KUKA KRL program: MyProgram_099().src

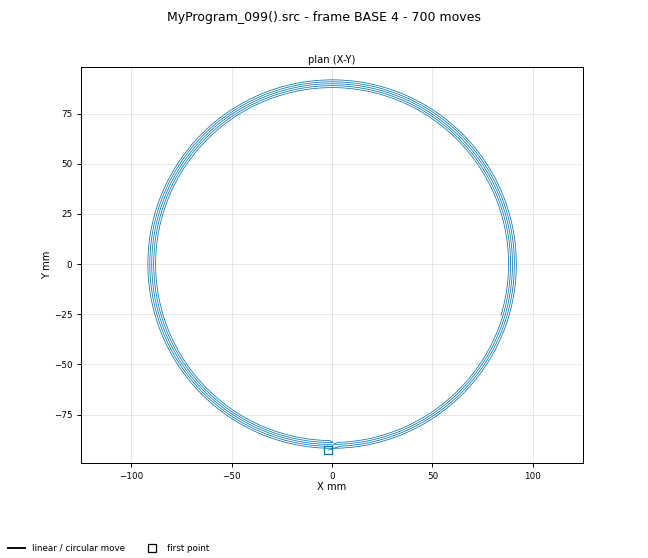
[picture p0: tool path of MyProgram_099().src in frame BASE 4, 700 of 700 moves have a stored position in this frame; points joined in program order, loops and branches not executed]
&ACCESS RVP
&REL 1
&PARAM TEMPLATE = C:\KRC\Roboter\Template\vorgabe
&PARAM EDITMASK = *
DEF MyProgram_099()
; ---- Setting reference (Base) ----
$BASE = BASE_DATA[4]

; --------------------------
; ---- Setting tool (TCP) ----
$TOOL = TOOL_DATA[3]
; --------------------------

$VEL.CP = VEL_APROX_PRINT
Startdeposition()
$VEL.CP = VEL_PRINT
LIN {X -1.871,Y -92.7683,Z 91,A -94.8232,B 24.9323,C -1.9,E1 24.9994,E2 179.961} C_DIS
Enddeposition()
LIN {X 0.618,Y -91.7983,Z 91,A -93.6423,B 24.932,C -1.905,E1 25.0028,E2 178.7684} C_DIS
Startdeposition()
$VEL.CP = VEL_PRINT
LIN {X -1.6204,Y -91.8049,Z 91,A -96.9281,B 24.9365,C -1.8408,E1 24.9932,E2 182.2064} C_DIS
LIN {X -6.6476,Y -91.5793,Z 91,A -99.0466,B 24.9341,C -1.8746,E1 24.9875,E2 184.2456} C_DIS
LIN {X -12.2271,Y -91.0017,Z 91,A -103.2009,B 24.9356,C -1.8535,E1 24.9758,E2 188.4527} C_DIS
LIN {X -15.9011,Y -90.4321,Z 91,A -104.6147,B 24.9335,C -1.8841,E1 24.9721,E2 189.7952} C_DIS
LIN {X -18.2695,Y -89.9835,Z 91,A -106.7072,B 24.9348,C -1.8652,E1 24.9662,E2 191.9348} C_DIS
LIN {X -22.9812,Y -88.8968,Z 91,A -109.6487,B 24.9345,C -1.8693,E1 24.9583,E2 194.8706} C_DIS
LIN {X -27.0599,Y -87.7413,Z 91,A -111.9748,B 24.9336,C -1.8816,E1 24.9521,E2 197.1715} C_DIS
LIN {X -31.2211,Y -86.3485,Z 91,A -114.7916,B 24.9336,C -1.8813,E1 24.9447,E2 199.9944} C_DIS
LIN {X -34.2722,Y -85.1832,Z 91,A -116.9435,B 24.9338,C -1.8795,E1 24.939,E2 202.1551} C_DIS
LIN {X -37.6537,Y -83.7434,Z 91,A -119.5434,B 24.9343,C -1.8722,E1 24.9323,E2 204.7786} C_DIS
LIN {X -42.2252,Y -81.5349,Z 91,A -122.8582,B 24.9343,C -1.8714,E1 24.9241,E2 208.1042} C_DIS
LIN {X -45.2073,Y -79.9207,Z 91,A -124.3084,B 24.9326,C -1.8955,E1 24.9206,E2 209.5014} C_DIS
LIN {X -48.7304,Y -77.8211,Z 91,A -127.0637,B 24.9328,C -1.893,E1 24.914,E2 212.271} C_DIS
LIN {X -51.619,Y -75.9359,Z 91,A -129.5861,B 24.9334,C -1.8847,E1 24.9081,E2 214.8214} C_DIS
LIN {X -54.5175,Y -73.8832,Z 91,A -131.4951,B 24.9325,C -1.8981,E1 24.9039,E2 216.7051} C_DIS
LIN {X -58.7556,Y -70.5588,Z 91,A -134.6797,B 24.9316,C -1.9098,E1 24.8969,E2 219.8739} C_DIS
LIN {X -60.9727,Y -68.6527,Z 91,A -136.6778,B 24.9318,C -1.9079,E1 24.8927,E2 221.8844} C_DIS
LIN {X -64.9121,Y -64.9421,Z 91,A -140.0394,B 24.9312,C -1.9153,E1 24.8859,E2 225.2422} C_DIS
LIN {X -67.1815,Y -62.5906,Z 91,A -142.1304,B 24.931,C -1.9181,E1 24.8819,E2 227.3356} C_DIS
LIN {X -70.739,Y -58.5387,Z 91,A -145.139,B 24.9297,C -1.9368,E1 24.8765,E2 230.3132} C_DIS
LIN {X -72.1644,Y -56.7724,Z 91,A -146.9681,B 24.9304,C -1.9274,E1 24.8732,E2 232.1734} C_DIS
LIN {X -75.8177,Y -51.7933,Z 91,A -150.4821,B 24.9289,C -1.9474,E1 24.8675,E2 235.657} C_DIS
LIN {X -77.8299,Y -48.7162,Z 91,A -153.8723,B 24.9309,C -1.92,E1 24.8623,E2 239.1296} C_DIS
LIN {X -80.0718,Y -44.9366,Z 91,A -155.5096,B 24.9279,C -1.9607,E1 24.8602,E2 240.6782} C_DIS
LIN {X -82.9877,Y -39.291,Z 91,A -159.9053,B 24.9281,C -1.9585,E1 24.8546,E2 245.1028} C_DIS
LIN {X -84.5445,Y -35.8192,Z 91,A -162.2753,B 24.9276,C -1.9654,E1 24.8519,E2 247.4694} C_DIS
LIN {X -86.3463,Y -31.2273,Z 91,A -165.1608,B 24.9265,C -1.9802,E1 24.8491,E2 250.3359} C_DIS
LIN {X -87.3543,Y -28.2838,Z 91,A -167.9303,B 24.9279,C -1.9612,E1 24.8466,E2 253.1666} C_DIS
LIN {X -88.49,Y -24.5019,Z 91,A -169.5246,B 24.9254,C -1.9946,E1 24.8454,E2 254.6904} C_DIS
LIN {X -89.3909,Y -20.979,Z 91,A -172.0935,B 24.9256,C -1.9925,E1 24.8437,E2 257.2792} C_DIS
LIN {X -90.1571,Y -17.3912,Z 91,A -174.3422,B 24.9249,C -2.0008,E1 24.8424,E2 259.5214} C_DIS
LIN {X -90.8192,Y -13.5236,Z 91,A -176.8189,B 24.9244,C -2.0076,E1 24.8413,E2 261.9966} C_DIS
LIN {X -91.1749,Y -10.8598,Z 91,A -178.5376,B 24.9241,C -2.0117,E1 24.8407,E2 263.716} C_DIS
LIN {X -91.5267,Y -7.3223,Z 91,A 179.3238,B 24.9234,C -2.0211,E1 24.8402,E2 265.8449} C_DIS
LIN {X -91.7396,Y -3.824,Z 91,A 177.0719,B 24.923,C -2.0261,E1 24.8399,E2 268.0983} C_DIS
LIN {X -91.8155,Y -0.8782,Z 91,A 175.1478,B 24.9228,C -2.0294,E1 24.8398,E2 270.0261} C_DIS
LIN {X -91.7727,Y 2.9233,Z 91,A 172.771,B 24.9222,C -2.0369,E1 24.8399,E2 272.3994} C_DIS
LIN {X -91.5374,Y 7.1893,Z 91,A 169.952,B 24.9219,C -2.0409,E1 24.8404,E2 275.2257} C_DIS
LIN {X -91.1985,Y 10.6584,Z 91,A 167.9398,B 24.921,C -2.0527,E1 24.841,E2 277.2218} C_DIS
LIN {X -90.6942,Y 14.3323,Z 91,A 165.6777,B 24.9203,C -2.0617,E1 24.842,E2 279.4761} C_DIS
LIN {X -90.1147,Y 17.6113,Z 91,A 163.4344,B 24.9202,C -2.0634,E1 24.8431,E2 281.7286} C_DIS
LIN {X -88.9887,Y 22.6236,Z 91,A 160.5247,B 24.9187,C -2.0823,E1 24.8449,E2 284.6101} C_DIS
LIN {X -88.2612,Y 25.3131,Z 91,A 158.5023,B 24.9189,C -2.0793,E1 24.8465,E2 286.6515} C_DIS
LIN {X -86.9975,Y 29.3631,Z 91,A 155.3931,B 24.9193,C -2.0739,E1 24.8492,E2 289.7914} C_DIS
LIN {X -85.8688,Y 32.5163,Z 91,A 154.1404,B 24.9169,C -2.1052,E1 24.8503,E2 290.9765} C_DIS
LIN {X -85.0065,Y 34.7084,Z 91,A 151.2137,B 24.9199,C -2.0665,E1 24.8536,E2 294.0118} C_DIS
LIN {X -82.8239,Y 39.6354,Z 91,A 149.1226,B 24.9162,C -2.1142,E1 24.8559,E2 296.0005} C_DIS
LIN {X -81.6777,Y 41.947,Z 91,A 147.2257,B 24.9165,C -2.1103,E1 24.8583,E2 297.9169} C_DIS
LIN {X -79.0825,Y 46.6554,Z 91,A 143.9691,B 24.9155,C -2.123,E1 24.8627,E2 301.1604} C_DIS
LIN {X -76.1928,Y 51.2397,Z 91,A 140.5759,B 24.9147,C -2.1321,E1 24.8679,E2 304.549} C_DIS
LIN {X -73.3066,Y 55.2895,Z 91,A 137.3458,B 24.9144,C -2.1366,E1 24.8732,E2 307.7838} C_DIS
LIN {X -69.6332,Y 59.851,Z 91,A 134.0172,B 24.9128,C -2.156,E1 24.879,E2 311.0817} C_DIS
LIN {X -67.3029,Y 62.4597,Z 91,A 131.7335,B 24.9126,C -2.1584,E1 24.8833,E2 313.3699} C_DIS
LIN {X -65.444,Y 64.404,Z 91,A 129.8568,B 24.9128,C -2.1565,E1 24.8869,E2 315.2593} C_DIS
LIN {X -62.1113,Y 67.6236,Z 91,A 127.3843,B 24.9112,C -2.1761,E1 24.8918,E2 317.6952} C_DIS
LIN {X -59.1378,Y 70.2397,Z 91,A 124.4002,B 24.912,C -2.1659,E1 24.8982,E2 320.7153} C_DIS
LIN {X -56.3727,Y 72.4779,Z 91,A 121.6226,B 24.913,C -2.1536,E1 24.9044,E2 323.5324} C_DIS
LIN {X -53.4479,Y 74.6599,Z 91,A 119.949,B 24.9111,C -2.1767,E1 24.9081,E2 325.1569} C_DIS
LIN {X -49.435,Y 77.3756,Z 91,A 116.84,B 24.9109,C -2.1799,E1 24.9153,E2 328.2685} C_DIS
LIN {X -44.1429,Y 80.513,Z 91,A 113.2762,B 24.9096,C -2.1953,E1 24.9238,E2 331.8064} C_DIS
LIN {X -41.9976,Y 81.6518,Z 91,A 111.4688,B 24.9101,C -2.1887,E1 24.9283,E2 333.6345} C_DIS
LIN {X -38.7679,Y 83.2334,Z 91,A 108.7733,B 24.911,C -2.1781,E1 24.9352,E2 336.362} C_DIS
LIN {X -35.7147,Y 84.5885,Z 91,A 107.4169,B 24.9089,C -2.2039,E1 24.9386,E2 337.6602} C_DIS
LIN {X -31.6123,Y 86.2055,Z 91,A 104.5487,B 24.9089,C -2.2039,E1 24.9461,E2 340.5344} C_DIS
LIN {X -29.457,Y 86.9656,Z 91,A 102.41,B 24.9106,C -2.1832,E1 24.9518,E2 342.7265} C_DIS
LIN {X -25.9931,Y 88.0632,Z 91,A 100.6921,B 24.909,C -2.203,E1 24.9563,E2 344.4001} C_DIS
LIN {X -22.5168,Y 89.0161,Z 91,A 98.4003,B 24.9089,C -2.2039,E1 24.9625,E2 346.6932} C_DIS
LIN {X -17.696,Y 90.0984,Z 91,A 95.646,B 24.9078,C -2.2172,E1 24.9699,E2 349.4195} C_DIS
LIN {X -13.9628,Y 90.7513,Z 91,A 92.1983,B 24.9105,C -2.1842,E1 24.9797,E2 352.9488} C_DIS
LIN {X -9.5944,Y 91.3165,Z 91,A 90.3815,B 24.9079,C -2.2156,E1 24.9845,E2 354.692} C_DIS
LIN {X -7.0102,Y 91.5516,Z 91,A 87.5465,B 24.9111,C -2.1772,E1 24.9927,E2 357.6194} C_DIS
LIN {X -1.6648,Y 91.8041,Z 91,A 84.4297,B 24.9104,C -2.1852,E1 25.0013,E2 360.7175} C_DIS
LIN {X 2.9296,Y 91.7725,Z 91,A 82.8065,B 24.907,C -2.2261,E1 25.0056,E2 362.2432} C_DIS
LIN {X 5.2509,Y 91.6691,Z 91,A 80.5872,B 24.9091,C -2.2008,E1 25.0119,E2 364.5218} C_DIS
LIN {X 10.4898,Y 91.2182,Z 91,A 77.508,B 24.9086,C -2.2071,E1 25.0204,E2 367.5842} C_DIS
LIN {X 14.3424,Y 90.6926,Z 91,A 75.2122,B 24.9083,C -2.2107,E1 25.0267,E2 369.8692} C_DIS
LIN {X 17.7373,Y 90.0905,Z 91,A 73.0288,B 24.9085,C -2.2088,E1 25.0327,E2 372.0547} C_DIS
LIN {X 20.9469,Y 89.3984,Z 91,A 71.1006,B 24.9082,C -2.2118,E1 25.038,E2 373.9732} C_DIS
LIN {X 24.2742,Y 88.5526,Z 91,A 69.1138,B 24.9079,C -2.2157,E1 25.0433,E2 375.9477} C_DIS
LIN {X 28.1738,Y 87.39,Z 91,A 66.5053,B 24.9083,C -2.2115,E1 25.0503,E2 378.5616} C_DIS
LIN {X 31.0195,Y 86.4215,Z 91,A 64.3973,B 24.9091,C -2.202,E1 25.0559,E2 380.6879} C_DIS
LIN {X 34.6134,Y 85.0451,Z 91,A 61.6457,B 24.9102,C -2.1877,E1 25.0631,E2 383.4671} C_DIS
LIN {X 37.6375,Y 83.7507,Z 91,A 60.1052,B 24.909,C -2.2028,E1 25.0669,E2 384.968} C_DIS
LIN {X 41.5759,Y 81.8665,Z 91,A 56.8355,B 24.9108,C -2.1808,E1 25.0752,E2 388.281} C_DIS
LIN {X 44.6417,Y 80.2365,Z 91,A 55.1885,B 24.9096,C -2.1957,E1 25.0792,E2 389.8882} C_DIS
LIN {X 47.7013,Y 78.456,Z 91,A 52.9995,B 24.9098,C -2.1931,E1 25.0844,E2 392.0764} C_DIS
LIN {X 51.4827,Y 76.0282,Z 91,A 50.2899,B 24.9098,C -2.192,E1 25.0907,E2 394.7798} C_DIS
LIN {X 55.1697,Y 73.3966,Z 91,A 47.5107,B 24.9101,C -2.1888,E1 25.097,E2 397.5568} C_DIS
LIN {X 57.5121,Y 71.577,Z 91,A 45.4868,B 24.9109,C -2.1793,E1 25.1015,E2 399.5955} C_DIS
LIN {X 60.3092,Y 69.2356,Z 91,A 42.9874,B 24.9119,C -2.1671,E1 25.1068,E2 402.114} C_DIS
LIN {X 64.3165,Y 65.5304,Z 91,A 39.985,B 24.9113,C -2.1743,E1 25.1129,E2 405.0871} C_DIS
LIN {X 66.3986,Y 63.4201,Z 91,A 37.8391,B 24.9125,C -2.1598,E1 25.1171,E2 407.2579} C_DIS
LIN {X 69.6395,Y 59.8436,Z 91,A 35.2905,B 24.9117,C -2.1695,E1 25.1217,E2 409.7723} C_DIS
LIN {X 71.1807,Y 58.0011,Z 91,A 33.5418,B 24.9127,C -2.1571,E1 25.1249,E2 411.5424} C_DIS
LIN {X 73.521,Y 55.0042,Z 91,A 31.1329,B 24.9133,C -2.15,E1 25.129,E2 413.9564} C_DIS
LIN {X 76.7059,Y 50.4675,Z 91,A 27.727,B 24.9138,C -2.1432,E1 25.1344,E2 417.3617} C_DIS
LIN {X 78.5486,Y 47.5489,Z 91,A 25.5473,B 24.9144,C -2.1366,E1 25.1376,E2 419.5458} C_DIS
LIN {X 80.3597,Y 44.4207,Z 91,A 23.3059,B 24.9148,C -2.1311,E1 25.1407,E2 421.7887} C_DIS
LIN {X 81.7511,Y 41.8032,Z 91,A 21.5002,B 24.9151,C -2.1276,E1 25.143,E2 423.5932} C_DIS
LIN {X 84.0935,Y 36.8644,Z 91,A 18.367,B 24.9151,C -2.128,E1 25.1467,E2 426.7084} C_DIS
LIN {X 85.7886,Y 32.7279,Z 91,A 15.2831,B 24.9166,C -2.1092,E1 25.1499,E2 429.8196} C_DIS
LIN {X 87.0104,Y 29.3248,Z 91,A 12.6948,B 24.918,C -2.0906,E1 25.1523,E2 432.4373} C_DIS
LIN {X 88.4115,Y 24.7837,Z 91,A 10.1763,B 24.9175,C -2.0978,E1 25.1542,E2 434.9244} C_DIS
LIN {X 89.2668,Y 21.4986,Z 91,A 8.0617,B 24.918,C -2.0915,E1 25.1557,E2 437.0417} C_DIS
LIN {X 90.0292,Y 18.0432,Z 91,A 6.1058,B 24.9178,C -2.0938,E1 25.1568,E2 438.9807} C_DIS
LIN {X 90.5062,Y 15.4757,Z 91,A 3.585,B 24.9207,C -2.0563,E1 25.1581,E2 441.5752} C_DIS
LIN {X 91.0927,Y 11.5308,Z 91,A 1.0412,B 24.9215,C -2.0465,E1 25.1589,E2 444.1271} C_DIS
LIN {X 91.5268,Y 7.321,Z 91,A -0.8141,B 24.9199,C -2.0667,E1 25.1594,E2 445.9239} C_DIS
LIN {X 91.8164,Y 0.7034,Z 91,A -5.665,B 24.9229,C -2.0273,E1 25.1598,E2 450.8387} C_DIS
LIN {X 91.7531,Y -3.4995,Z 91,A -7.5622,B 24.9216,C -2.0453,E1 25.1596,E2 452.6822} C_DIS
LIN {X 91.634,Y -5.8342,Z 91,A -9.8304,B 24.9242,C -2.0111,E1 25.1592,E2 455.0176} C_DIS
LIN {X 91.2306,Y -10.3843,Z 91,A -12.4103,B 24.9242,C -2.0118,E1 25.1584,E2 457.5807} C_DIS
LIN {X 90.7427,Y -14.0184,Z 91,A -13.6348,B 24.9217,C -2.0434,E1 25.1579,E2 458.7235} C_DIS
LIN {X 90.1084,Y -17.6439,Z 91,A -16.425,B 24.9237,C -2.0179,E1 25.1565,E2 461.5575} C_DIS
LIN {X 89.3627,Y -21.0966,Z 91,A -18.8721,B 24.9248,C -2.002,E1 25.155,E2 464.0279} C_DIS
LIN {X 88.3779,Y -24.9022,Z 91,A -21.0609,B 24.9248,C -2.0039,E1 25.1534,E2 466.1996} C_DIS
LIN {X 87.2223,Y -28.688,Z 91,A -24.2136,B 24.9271,C -1.9714,E1 25.1506,E2 469.4112} C_DIS
LIN {X 85.7809,Y -32.7483,Z 91,A -27.2588,B 24.9287,C -1.9503,E1 25.1475,E2 472.4892} C_DIS
LIN {X 83.6294,Y -37.9068,Z 91,A -29.6005,B 24.9264,C -1.9812,E1 25.145,E2 474.7453} C_DIS
LIN {X 81.4119,Y -42.4605,Z 91,A -32.73,B 24.927,C -1.9729,E1 25.1411,E2 477.8775} C_DIS
LIN {X 79.2087,Y -46.4419,Z 91,A -35.5915,B 24.9277,C -1.9639,E1 25.1372,E2 480.7456} C_DIS
LIN {X 76.6368,Y -50.5723,Z 91,A -38.5481,B 24.9281,C -1.9582,E1 25.1328,E2 483.7007} C_DIS
LIN {X 74.7848,Y -53.2729,Z 91,A -41.3625,B 24.9305,C -1.9248,E1 25.1281,E2 486.5802} C_DIS
LIN {X 72.2029,Y -56.7237,Z 91,A -43.3164,B 24.9291,C -1.944,E1 25.1249,E2 488.4795} C_DIS
LIN {X 68.8101,Y -60.7963,Z 91,A -46.5699,B 24.9296,C -1.9374,E1 25.119,E2 491.7338} C_DIS
LIN {X 65.1686,Y -64.6827,Z 91,A -49.7372,B 24.9298,C -1.9348,E1 25.1129,E2 494.8936} C_DIS
LIN {X 61.0956,Y -68.5429,Z 91,A -52.8337,B 24.9294,C -1.9411,E1 25.1067,E2 497.9624} C_DIS
LIN {X 57.1312,Y -71.8807,Z 91,A -56.2409,B 24.9303,C -1.9276,E1 25.0994,E2 501.3884} C_DIS
LIN {X 52.9571,Y -75.0095,Z 91,A -59.5776,B 24.9311,C -1.9178,E1 25.0919,E2 504.7363} C_DIS
LIN {X 50.7563,Y -76.5155,Z 91,A -61.9567,B 24.9331,C -1.8891,E1 25.0862,E2 507.1751} C_DIS
LIN {X 47.9378,Y -78.3123,Z 91,A -63.7712,B 24.9327,C -1.8948,E1 25.0819,E2 508.9706} C_DIS
LIN {X 45.3567,Y -79.8355,Z 91,A -65.8478,B 24.9335,C -1.8841,E1 25.0768,E2 511.0661} C_DIS
LIN {X 41.0102,Y -82.1522,Z 91,A -68.696,B 24.9333,C -1.8869,E1 25.0698,E2 513.8999} C_DIS
LIN {X 37.6512,Y -83.7445,Z 91,A -71.5601,B 24.9348,C -1.8644,E1 25.0624,E2 516.81} C_DIS
LIN {X 33.6749,Y -85.4206,Z 91,A -73.3515,B 24.9329,C -1.8919,E1 25.0579,E2 518.5323} C_DIS
LIN {X 30.9775,Y -86.4364,Z 91,A -75.7123,B 24.9344,C -1.87,E1 25.0516,E2 520.9401} C_DIS
LIN {X 27.9319,Y -87.4682,Z 91,A -77.5636,B 24.9342,C -1.873,E1 25.0467,E2 522.7809} C_DIS
LIN {X 23.4924,Y -88.7634,Z 91,A -79.9052,B 24.9331,C -1.8886,E1 25.0405,E2 525.0815} C_DIS
LIN {X 21.0845,Y -89.3658,Z 91,A -81.7171,B 24.9339,C -1.878,E1 25.0356,E2 526.916} C_DIS
LIN {X 17.6018,Y -90.1166,Z 91,A -83.903,B 24.9339,C -1.8774,E1 25.0296,E2 529.1007} C_DIS
LIN {X 14.172,Y -90.719,Z 91,A -86.8872,B 24.936,C -1.8482,E1 25.0212,E2 532.1511} C_DIS
LIN {X 9.7533,Y -91.2999,Z 91,A -89.1415,B 24.9348,C -1.8643,E1 25.015,E2 534.3656} C_DIS
LIN {X 4.5778,Y -91.7055,Z 91,A -91.9372,B 24.9339,C -1.8779,E1 25.0073,E2 537.1278} C_DIS
LIN {X 0.618,Y -91.7983,Z 91,A -93.6392,B 24.9321,C -1.9036,E1 25.0028,E2 538.7683} C_DIS
Enddeposition()
LIN {X 0.618,Y -91.7983,Z 91,A -93.6392,B 24.9321,C -1.9036,E1 25.0028,E2 538.7683} C_DIS
Startdeposition()
$VEL.CP = VEL_PRINT
LIN {X 4.1584,Y -90.756,Z 91,A -91.557,B 24.9312,C -1.9156,E1 25.0086,E2 536.6583} C_DIS
LIN {X 9.1157,Y -90.3931,Z 91,A -88.3749,B 24.931,C -1.9187,E1 25.0175,E2 533.4704} C_DIS
LIN {X 13.9356,Y -89.7761,Z 91,A -85.2695,B 24.9307,C -1.9221,E1 25.0261,E2 530.3596} C_DIS
LIN {X 17.0007,Y -89.2466,Z 91,A -83.4033,B 24.9309,C -1.9204,E1 25.0312,E2 528.4996} C_DIS
LIN {X 20.0337,Y -88.6152,Z 91,A -81.2501,B 24.9302,C -1.9291,E1 25.0371,E2 526.3286} C_DIS
LIN {X 23.2381,Y -87.8295,Z 91,A -78.8258,B 24.9292,C -1.9432,E1 25.0438,E2 523.8747} C_DIS
LIN {X 27.6774,Y -86.5333,Z 91,A -75.8242,B 24.9287,C -1.9496,E1 25.0518,E2 520.8633} C_DIS
LIN {X 30.8475,Y -85.4545,Z 91,A -74.1343,B 24.9296,C -1.9375,E1 25.0562,E2 519.2055} C_DIS
LIN {X 33.3178,Y -84.5215,Z 91,A -71.8666,B 24.9279,C -1.9611,E1 25.0622,E2 516.887} C_DIS
LIN {X 37.0033,Y -82.974,Z 91,A -69.8491,B 24.9289,C -1.947,E1 25.0672,E2 514.9078} C_DIS
LIN {X 40.7457,Y -81.2026,Z 91,A -67.4571,B 24.9292,C -1.9434,E1 25.0732,E2 512.5306} C_DIS
LIN {X 45.8988,Y -78.4054,Z 91,A -63.8067,B 24.9288,C -1.9482,E1 25.0821,E2 508.8795} C_DIS
LIN {X 48.4739,Y -76.8389,Z 91,A -61.3161,B 24.927,C -1.9729,E1 25.0881,E2 506.3385} C_DIS
LIN {X 51.4708,Y -74.8661,Z 91,A -59.7361,B 24.9285,C -1.9529,E1 25.0917,E2 504.8111} C_DIS
LIN {X 53.231,Y -73.6242,Z 91,A -57.7606,B 24.9267,C -1.9779,E1 25.0963,E2 502.7836} C_DIS
LIN {X 55.9408,Y -71.5878,Z 91,A -55.9636,B 24.9272,C -1.9702,E1 25.1002,E2 501.0114} C_DIS
LIN {X 59.5061,Y -68.6518,Z 91,A -53.2212,B 24.9272,C -1.9706,E1 25.106,E2 498.2786} C_DIS
LIN {X 62.6549,Y -65.7896,Z 91,A -50.4558,B 24.9265,C -1.9798,E1 25.1117,E2 495.5026} C_DIS
LIN {X 65.6688,Y -62.782,Z 91,A -47.6399,B 24.9257,C -1.9911,E1 25.1172,E2 492.672} C_DIS
LIN {X 68.6181,Y -59.5448,Z 91,A -44.9149,B 24.9252,C -1.9968,E1 25.1223,E2 489.9459} C_DIS
LIN {X 71.4759,Y -56.0825,Z 91,A -42.363,B 24.9254,C -1.9941,E1 25.1267,E2 487.4122} C_DIS
LIN {X 73.3997,Y -53.5393,Z 91,A -40.0493,B 24.9242,C -2.0106,E1 25.1306,E2 485.0707} C_DIS
LIN {X 75.1288,Y -51.0847,Z 91,A -37.9428,B 24.9232,C -2.0237,E1 25.1339,E2 482.9436} C_DIS
LIN {X 76.9734,Y -48.2605,Z 91,A -36.2432,B 24.9239,C -2.014,E1 25.1364,E2 481.2755} C_DIS
LIN {X 80.0841,Y -42.9025,Z 91,A -32.5835,B 24.9238,C -2.0162,E1 25.1415,E2 477.6295} C_DIS
LIN {X 81.76,Y -39.6142,Z 91,A -29.8596,B 24.9221,C -2.0377,E1 25.1449,E2 474.8696} C_DIS
LIN {X 84.0612,Y -34.4616,Z 91,A -26.4028,B 24.9216,C -2.0447,E1 25.1487,E2 471.415} C_DIS
LIN {X 85.537,Y -30.6176,Z 91,A -23.7834,B 24.9209,C -2.0536,E1 25.1512,E2 468.7894} C_DIS
LIN {X 86.9984,Y -26.1775,Z 91,A -21.0593,B 24.9209,C -2.0545,E1 25.1535,E2 466.0786} C_DIS
LIN {X 87.7401,Y -23.5719,Z 91,A -18.6737,B 24.9185,C -2.085,E1 25.1553,E2 463.6348} C_DIS
LIN {X 88.7223,Y -19.5538,Z 91,A -17.0645,B 24.9207,C -2.0563,E1 25.1562,E2 462.1027} C_DIS
LIN {X 89.664,Y -14.6436,Z 91,A -13.7979,B 24.9196,C -2.0705,E1 25.1579,E2 458.8217} C_DIS
LIN {X 90.2499,Y -10.4366,Z 91,A -10.2257,B 24.9163,C -2.1122,E1 25.1591,E2 455.1722} C_DIS
LIN {X 90.6461,Y -6.1026,Z 91,A -8.3392,B 24.9181,C -2.0891,E1 25.1595,E2 453.3513} C_DIS
LIN {X 90.8502,Y 0.3857,Z 91,A -4.6458,B 24.9183,C -2.0875,E1 25.1598,E2 449.6836} C_DIS
LIN {X 90.7295,Y 4.7113,Z 91,A -1.5248,B 24.9165,C -2.1106,E1 25.1595,E2 446.5267} C_DIS
LIN {X 90.4844,Y 8.1587,Z 91,A 1.1089,B 24.9146,C -2.1343,E1 25.1589,E2 443.8528} C_DIS
LIN {X 90.1376,Y 11.3689,Z 91,A 3.1047,B 24.9142,C -2.1392,E1 25.1582,E2 441.8571} C_DIS
LIN {X 89.4311,Y 16.0005,Z 91,A 5.6179,B 24.9147,C -2.1322,E1 25.157,E2 439.3753} C_DIS
LIN {X 88.7122,Y 19.5999,Z 91,A 7.9811,B 24.914,C -2.1411,E1 25.1557,E2 437.0048} C_DIS
LIN {X 87.8643,Y 23.1053,Z 91,A 10.175,B 24.9137,C -2.1451,E1 25.1542,E2 434.8141} C_DIS
LIN {X 87.0404,Y 26.0378,Z 91,A 12.9125,B 24.9108,C -2.1809,E1 25.1519,E2 432.0077} C_DIS
LIN {X 85.6391,Y 30.3304,Z 91,A 14.9002,B 24.9127,C -2.1577,E1 25.1502,E2 430.0859} C_DIS
LIN {X 84.3384,Y 33.7776,Z 91,A 17.4837,B 24.9114,C -2.174,E1 25.1475,E2 427.4784} C_DIS
LIN {X 81.8851,Y 39.3546,Z 91,A 21.0023,B 24.9114,C -2.173,E1 25.1435,E2 423.9811} C_DIS
LIN {X 80.457,Y 42.1974,Z 91,A 23.1119,B 24.9107,C -2.1823,E1 25.1408,E2 421.8608} C_DIS
LIN {X 78.6974,Y 45.3949,Z 91,A 25.3823,B 24.9103,C -2.1874,E1 25.1376,E2 419.5902} C_DIS
LIN {X 76.8297,Y 48.4904,Z 91,A 28.6177,B 24.9069,C -2.228,E1 25.1327,E2 416.2751} C_DIS
LIN {X 73.9523,Y 52.7733,Z 91,A 30.8168,B 24.9094,C -2.1979,E1 25.1293,E2 414.1578} C_DIS
LIN {X 72.4084,Y 54.8736,Z 91,A 32.7634,B 24.9082,C -2.2128,E1 25.126,E2 412.1854} C_DIS
LIN {X 69.6725,Y 58.3078,Z 91,A 35.0599,B 24.909,C -2.2024,E1 25.122,E2 409.9241} C_DIS
LIN {X 67.8377,Y 60.432,Z 91,A 37.5822,B 24.9064,C -2.2333,E1 25.1172,E2 407.34} C_DIS
LIN {X 65.2986,Y 63.167,Z 91,A 39.3801,B 24.9077,C -2.2185,E1 25.1138,E2 405.5847} C_DIS
LIN {X 62.0203,Y 66.3893,Z 91,A 42.8832,B 24.9054,C -2.246,E1 25.1066,E2 402.0312} C_DIS
LIN {X 59.0629,Y 69.0331,Z 91,A 44.733,B 24.9069,C -2.2278,E1 25.1029,E2 400.2319} C_DIS
LIN {X 56.3168,Y 71.2907,Z 91,A 46.6902,B 24.9074,C -2.2219,E1 25.0986,E2 398.2958} C_DIS
LIN {X 51.9296,Y 74.5472,Z 91,A 50.3063,B 24.9064,C -2.2338,E1 25.0905,E2 394.6645} C_DIS
LIN {X 49.3768,Y 76.2628,Z 91,A 52.6957,B 24.9048,C -2.2526,E1 25.0848,E2 392.2385} C_DIS
LIN {X 45.2588,Y 78.7756,Z 91,A 55.1567,B 24.9061,C -2.2368,E1 25.079,E2 389.8225} C_DIS
LIN {X 42.6907,Y 80.1965,Z 91,A 57.8766,B 24.9034,C -2.2695,E1 25.0721,E2 387.0329} C_DIS
LIN {X 39.077,Y 82.0177,Z 91,A 59.7136,B 24.9052,C -2.2478,E1 25.0677,E2 385.2522} C_DIS
LIN {X 36.3863,Y 83.2466,Z 91,A 61.8564,B 24.9042,C -2.2594,E1 25.0621,E2 383.0871} C_DIS
LIN {X 31.1137,Y 85.3574,Z 91,A 65.2141,B 24.9046,C -2.2552,E1 25.0534,E2 379.7467} C_DIS
LIN {X 24.766,Y 87.4105,Z 91,A 69.073,B 24.9053,C -2.2465,E1 25.0432,E2 375.9152} C_DIS
LIN {X 21.9648,Y 88.1564,Z 91,A 71.0348,B 24.9048,C -2.2522,E1 25.0379,E2 373.9432} C_DIS
LIN {X 19.8013,Y 88.6675,Z 91,A 72.6535,B 24.9042,C -2.2602,E1 25.0334,E2 372.3077} C_DIS
LIN {X 16.1221,Y 89.4093,Z 91,A 74.9076,B 24.9044,C -2.2574,E1 25.0273,E2 370.063} C_DIS
LIN {X 12.6752,Y 89.9628,Z 91,A 77.1902,B 24.9041,C -2.2607,E1 25.021,E2 367.7745} C_DIS
LIN {X 10.0015,Y 90.299,Z 91,A 79.5672,B 24.9022,C -2.2837,E1 25.0142,E2 365.3446} C_DIS
LIN {X 5.8925,Y 90.6601,Z 91,A 81.4832,B 24.9041,C -2.2608,E1 25.009,E2 363.4838} C_DIS
LIN {X 1.9282,Y 90.8312,Z 91,A 84.5611,B 24.9025,C -2.2797,E1 25.0003,E2 360.3617} C_DIS
LIN {X -1.7935,Y 90.8336,Z 91,A 87.1248,B 24.9019,C -2.2863,E1 24.9931,E2 357.7822} C_DIS
LIN {X -6.2609,Y 90.6354,Z 91,A 89.1872,B 24.9042,C -2.2601,E1 24.9875,E2 355.7811} C_DIS
LIN {X -9.6513,Y 90.3374,Z 91,A 91.6381,B 24.9034,C -2.269,E1 24.9807,E2 353.3078} C_DIS
LIN {X -14.4111,Y 89.7026,Z 91,A 94.3867,B 24.9044,C -2.2578,E1 24.9731,E2 350.5833} C_DIS
LIN {X -17.7736,Y 89.0962,Z 91,A 96.5497,B 24.9044,C -2.2564,E1 24.9672,E2 348.4214} C_DIS
LIN {X -22.5609,Y 88.0055,Z 91,A 99.6178,B 24.9048,C -2.2526,E1 24.9589,E2 345.3582} C_DIS
LIN {X -25.9023,Y 87.0806,Z 91,A 102.3517,B 24.9035,C -2.2678,E1 24.9515,E2 342.5836} C_DIS
LIN {X -29.4083,Y 85.96,Z 91,A 103.9465,B 24.9057,C -2.2418,E1 24.9474,E2 341.0478} C_DIS
LIN {X -34.598,Y 84.0056,Z 91,A 107.537,B 24.9059,C -2.24,E1 24.938,E2 337.4538} C_DIS
LIN {X -38.7521,Y 82.1722,Z 91,A 110.5902,B 24.9057,C -2.2417,E1 24.9302,E2 334.3891} C_DIS
LIN {X -42.2812,Y 80.413,Z 91,A 112.8737,B 24.9066,C -2.2313,E1 24.9246,E2 332.1243} C_DIS
LIN {X -45.3884,Y 78.7011,Z 91,A 115.7017,B 24.9054,C -2.2459,E1 24.9176,E2 329.2532} C_DIS
LIN {X -48.2393,Y 76.9866,Z 91,A 117.3208,B 24.907,C -2.227,E1 24.9139,E2 327.674} C_DIS
LIN {X -51.8616,Y 74.5944,Z 91,A 119.9123,B 24.9078,C -2.2171,E1 24.9079,E2 325.0975} C_DIS
LIN {X -57.0402,Y 70.7136,Z 91,A 123.8053,B 24.909,C -2.2027,E1 24.8993,E2 321.2247} C_DIS
LIN {X -61.1023,Y 67.2358,Z 91,A 127.3282,B 24.9092,C -2.1997,E1 24.8918,E2 317.6952} C_DIS
LIN {X -64.599,Y 63.8822,Z 91,A 130.5798,B 24.9093,C -2.1984,E1 24.8853,E2 314.4331} C_DIS
LIN {X -68.5499,Y 59.623,Z 91,A 133.9788,B 24.9108,C -2.1812,E1 24.879,E2 311.0602} C_DIS
LIN {X -71.1685,Y 56.4712,Z 91,A 136.9376,B 24.9104,C -2.1858,E1 24.8737,E2 308.0766} C_DIS
LIN {X -72.5513,Y 54.6834,Z 91,A 139.0192,B 24.909,C -2.202,E1 24.8701,E2 305.9464} C_DIS
LIN {X -74.8868,Y 51.4409,Z 91,A 140.7233,B 24.9117,C -2.1703,E1 24.8675,E2 304.3097} C_DIS
LIN {X -76.9938,Y 48.2277,Z 91,A 143.2305,B 24.912,C -2.166,E1 24.8637,E2 301.8} C_DIS
LIN {X -78.3435,Y 46.0035,Z 91,A 145.1627,B 24.9117,C -2.1701,E1 24.8609,E2 299.8479} C_DIS
LIN {X -80.6948,Y 41.7422,Z 91,A 147.8799,B 24.9133,C -2.1506,E1 24.8573,E2 297.1631} C_DIS
LIN {X -81.654,Y 39.8318,Z 91,A 149.7881,B 24.9122,C -2.1635,E1 24.8549,E2 295.2138} C_DIS
LIN {X -84.201,Y 34.1198,Z 91,A 153.418,B 24.9139,C -2.1421,E1 24.851,E2 291.6149} C_DIS
LIN {X -85.4058,Y 30.981,Z 91,A 156.04,B 24.9132,C -2.1507,E1 24.8484,E2 288.9575} C_DIS
LIN {X -86.5082,Y 27.7549,Z 91,A 158.2305,B 24.9137,C -2.1452,E1 24.8465,E2 286.7675} C_DIS
LIN {X -87.5165,Y 24.3915,Z 91,A 159.6372,B 24.9162,C -2.114,E1 24.8455,E2 285.4273} C_DIS
LIN {X -88.7635,Y 19.3649,Z 91,A 163.4898,B 24.9156,C -2.1212,E1 24.843,E2 281.5348} C_DIS
LIN {X -89.5927,Y 15.07,Z 91,A 165.9906,B 24.9169,C -2.1047,E1 24.8418,E2 279.0587} C_DIS
LIN {X -90.1106,Y 11.5778,Z 91,A 168.0404,B 24.9179,C -2.0923,E1 24.841,E2 277.0262} C_DIS
LIN {X -90.5503,Y 7.3902,Z 91,A 171.4811,B 24.9167,C -2.1073,E1 24.8401,E2 273.529} C_DIS
LIN {X -90.7723,Y 3.7898,Z 91,A 173.2246,B 24.9186,C -2.084,E1 24.8399,E2 271.8306} C_DIS
LIN {X -90.8509,Y 0.2387,Z 91,A 175.328,B 24.9194,C -2.0728,E1 24.8398,E2 269.7413} C_DIS
LIN {X -90.7784,Y -3.6462,Z 91,A 178.2134,B 24.919,C -2.078,E1 24.84,E2 266.8261} C_DIS
LIN {X -90.49,Y -8.0942,Z 91,A -179.2177,B 24.9203,C -2.0618,E1 24.8406,E2 264.2805} C_DIS
LIN {X -90.1682,Y -11.1231,Z 91,A -177.1418,B 24.9203,C -2.0604,E1 24.8413,E2 262.1955} C_DIS
LIN {X -89.385,Y -16.2575,Z 91,A -173.9553,B 24.9214,C -2.0475,E1 24.8427,E2 259.0209} C_DIS
LIN {X -88.5582,Y -20.2836,Z 91,A -170.7525,B 24.9206,C -2.058,E1 24.8447,E2 255.7741} C_DIS
LIN {X -87.6125,Y -24.0427,Z 91,A -168.8693,B 24.9225,C -2.0335,E1 24.846,E2 253.9385} C_DIS
LIN {X -86.1262,Y -28.9179,Z 91,A -165.6669,B 24.9232,C -2.0235,E1 24.8487,E2 250.7414} C_DIS
LIN {X -84.7789,Y -32.6577,Z 91,A -163.109,B 24.9237,C -2.0178,E1 24.8512,E2 248.1828} C_DIS
LIN {X -83.3375,Y -36.1777,Z 91,A -160.8959,B 24.9246,C -2.0052,E1 24.8536,E2 245.9873} C_DIS
LIN {X -82.0258,Y -39.0601,Z 91,A -157.9149,B 24.9227,C -2.0298,E1 24.8572,E2 242.9314} C_DIS
LIN {X -79.9712,Y -43.1111,Z 91,A -155.867,B 24.9252,C -1.9968,E1 24.8598,E2 240.9514} C_DIS
LIN {X -77.9745,Y -46.627,Z 91,A -153.0803,B 24.9252,C -1.9973,E1 24.8637,E2 238.1491} C_DIS
LIN {X -75.6797,Y -50.2656,Z 91,A -150.7183,B 24.9265,C -1.9795,E1 24.8673,E2 235.8175} C_DIS
LIN {X -73.2075,Y -53.8019,Z 91,A -147.3017,B 24.9254,C -1.9944,E1 24.8729,E2 232.349} C_DIS
LIN {X -71.0578,Y -56.6114,Z 91,A -145.8352,B 24.9276,C -1.9653,E1 24.8754,E2 230.9449} C_DIS
LIN {X -67.0667,Y -61.2866,Z 91,A -141.6957,B 24.9276,C -1.9646,E1 24.883,E2 226.7884} C_DIS
LIN {X -64.65,Y -63.8304,Z 91,A -138.3628,B 24.9254,C -1.9953,E1 24.8897,E2 223.3681} C_DIS
LIN {X -60.6822,Y -67.6139,Z 91,A -136.0096,B 24.9285,C -1.9533,E1 24.8943,E2 221.1054} C_DIS
LIN {X -55.145,Y -72.2019,Z 91,A -131.4261,B 24.929,C -1.9464,E1 24.9043,E2 216.5211} C_DIS
LIN {X -53.0613,Y -73.7467,Z 91,A -129.9963,B 24.9297,C -1.937,E1 24.9074,E2 215.1086} C_DIS
LIN {X -48.4772,Y -76.838,Z 91,A -126.2545,B 24.9295,C -1.9396,E1 24.9162,E2 211.3483} C_DIS
LIN {X -46.4273,Y -78.0929,Z 91,A -123.787,B 24.9274,C -1.9682,E1 24.9224,E2 208.8052} C_DIS
LIN {X -41.9804,Y -80.5707,Z 91,A -121.4896,B 24.9299,C -1.9343,E1 24.9278,E2 206.5821} C_DIS
LIN {X -39.0898,Y -82.0116,Z 91,A -119.7231,B 24.9307,C -1.9232,E1 24.9322,E2 204.8375} C_DIS
LIN {X -33.8459,Y -84.3112,Z 91,A -115.9009,B 24.9304,C -1.9262,E1 24.942,E2 200.9993} C_DIS
LIN {X -27.7711,Y -86.5029,Z 91,A -112.0342,B 24.9312,C -1.9159,E1 24.9522,E2 197.1494} C_DIS
LIN {X -24.6763,Y -87.4359,Z 91,A -109.8697,B 24.931,C -1.9186,E1 24.958,E2 194.9748} C_DIS
LIN {X -22.4934,Y -88.0227,Z 91,A -107.7274,B 24.9293,C -1.9416,E1 24.964,E2 192.7748} C_DIS
LIN {X -18.7524,Y -88.8952,Z 91,A -105.9241,B 24.9309,C -1.9199,E1 24.9687,E2 191.0211} C_DIS
LIN {X -15.4888,Y -89.5226,Z 91,A -104.0263,B 24.9314,C -1.9125,E1 24.9739,E2 189.1387} C_DIS
LIN {X -11.6873,Y -90.0963,Z 91,A -100.9255,B 24.9298,C -1.9347,E1 24.9826,E2 185.9828} C_DIS
LIN {X -8.381,Y -90.4639,Z 91,A -99.3035,B 24.931,C -1.9185,E1 24.987,E2 184.3984} C_DIS
LIN {X -5.5622,Y -90.6818,Z 91,A -96.7656,B 24.9291,C -1.9441,E1 24.9943,E2 181.799} C_DIS
LIN {X -1.3183,Y -90.842,Z 91,A -95.384,B 24.9323,C -1.9005,E1 24.9979,E2 180.5205} C_DIS
LIN {X 0.6013,Y -90.8167,Z 91,A -93.5732,B 24.9308,C -1.9216,E1 25.0031,E2 178.6598} C_DIS
Enddeposition()
LIN {X 0.6013,Y -90.8167,Z 91,A -93.5732,B 24.9308,C -1.9216,E1 25.0031,E2 178.6598} C_DIS
Startdeposition()
$VEL.CP = VEL_PRINT
LIN {X -0.5524,Y -89.8817,Z 91,A -95.0568,B 24.9314,C -1.9126,E1 24.9989,E2 180.1648} C_DIS
LIN {X -4.4631,Y -89.7729,Z 91,A -97.6525,B 24.9317,C -1.9088,E1 24.9916,E2 182.7696} C_DIS
LIN {X -7.0973,Y -89.6027,Z 91,A -99.5036,B 24.9321,C -1.9033,E1 24.9864,E2 184.6345} C_DIS
LIN {X -11.147,Y -89.1901,Z 91,A -102.3407,B 24.9326,C -1.8958,E1 24.9785,E2 187.4913} C_DIS
LIN {X -13.9956,Y -88.7875,Z 91,A -104.0208,B 24.9322,C -1.9012,E1 24.9739,E2 189.16} C_DIS
LIN {X -17.3887,Y -88.1863,Z 91,A -106.2209,B 24.9322,C -1.9019,E1 24.9678,E2 191.3608} C_DIS
LIN {X -23.0107,Y -86.8885,Z 91,A -109.5869,B 24.9313,C -1.9138,E1 24.9587,E2 194.703} C_DIS
LIN {X -26.7459,Y -85.812,Z 91,A -111.9957,B 24.9311,C -1.9177,E1 24.9523,E2 197.1066} C_DIS
LIN {X -31.2905,Y -84.2608,Z 91,A -115.3495,B 24.9315,C -1.9109,E1 24.9434,E2 200.483} C_DIS
LIN {X -37.9027,Y -81.501,Z 91,A -119.6696,B 24.9306,C -1.9234,E1 24.9323,E2 204.7833} C_DIS
LIN {X -40.0466,Y -80.4693,Z 91,A -121.5905,B 24.9314,C -1.9126,E1 24.9274,E2 206.7351} C_DIS
LIN {X -46.3543,Y -77.0094,Z 91,A -125.9374,B 24.9304,C -1.9263,E1 24.9169,E2 211.062} C_DIS
LIN {X -52.0876,Y -73.2525,Z 91,A -130.379,B 24.9301,C -1.9309,E1 24.9066,E2 215.5072} C_DIS
LIN {X -54.3467,Y -71.5937,Z 91,A -133.6171,B 24.933,C -1.89,E1 24.8991,E2 218.8543} C_DIS
LIN {X -59.04,Y -67.7739,Z 91,A -136.1052,B 24.9295,C -1.9386,E1 24.8941,E2 221.2363} C_DIS
LIN {X -62.3159,Y -64.7746,Z 91,A -139.4066,B 24.9302,C -1.9301,E1 24.8873,E2 224.5714} C_DIS
LIN {X -65.7421,Y -61.2956,Z 91,A -142.926,B 24.9305,C -1.9247,E1 24.8805,E2 228.119} C_DIS
LIN {X -68.568,Y -58.1163,Z 91,A -144.8257,B 24.9283,C -1.9552,E1 24.8771,E2 229.9548} C_DIS
LIN {X -70.6554,Y -55.5597,Z 91,A -147.401,B 24.929,C -1.946,E1 24.8726,E2 232.5639} C_DIS
LIN {X -74.1635,Y -50.7834,Z 91,A -150.8192,B 24.9275,C -1.9661,E1 24.8671,E2 235.9511} C_DIS
LIN {X -76.0772,Y -47.8683,Z 91,A -153.4124,B 24.9279,C -1.9608,E1 24.8631,E2 238.5699} C_DIS
LIN {X -78.6373,Y -43.535,Z 91,A -156.4908,B 24.927,C -1.9732,E1 24.8589,E2 241.6348} C_DIS
LIN {X -81.1622,Y -38.6222,Z 91,A -159.8938,B 24.926,C -1.9865,E1 24.8547,E2 245.0246} C_DIS
LIN {X -82.6424,Y -35.3453,Z 91,A -162.1777,B 24.9255,C -1.9932,E1 24.8521,E2 247.3049} C_DIS
LIN {X -84.3858,Y -30.953,Z 91,A -165.1541,B 24.9248,C -2.003,E1 24.8491,E2 250.2746} C_DIS
LIN {X -85.479,Y -27.7918,Z 91,A -167.8988,B 24.9256,C -1.9916,E1 24.8467,E2 253.0625} C_DIS
LIN {X -86.569,Y -24.1855,Z 91,A -169.542,B 24.9234,C -2.0208,E1 24.8455,E2 254.6452} C_DIS
LIN {X -87.7476,Y -19.4807,Z 91,A -172.6074,B 24.9226,C -2.031,E1 24.8434,E2 257.7043} C_DIS
LIN {X -88.2836,Y -16.8829,Z 91,A -175.0876,B 24.924,C -2.0134,E1 24.8421,E2 260.2412} C_DIS
LIN {X -88.8965,Y -13.2902,Z 91,A -177.2895,B 24.9232,C -2.0241,E1 24.8412,E2 262.4307} C_DIS
LIN {X -89.4731,Y -8.5844,Z 91,A -179.9343,B 24.9216,C -2.0446,E1 24.8404,E2 265.0425} C_DIS
LIN {X -89.8173,Y -3.4685,Z 91,A 176.2871,B 24.9219,C -2.0403,E1 24.8398,E2 268.854} C_DIS
LIN {X -89.8838,Y -0.0645,Z 91,A 174.7112,B 24.9201,C -2.0644,E1 24.8398,E2 270.382} C_DIS
LIN {X -89.8298,Y 3.1122,Z 91,A 171.7987,B 24.9216,C -2.0454,E1 24.8401,E2 273.3574} C_DIS
LIN {X -89.5775,Y 7.4135,Z 91,A 169.5322,B 24.9198,C -2.0679,E1 24.8405,E2 275.5837} C_DIS
LIN {X -89.1188,Y 11.6982,Z 91,A 167.3191,B 24.9179,C -2.0921,E1 24.8412,E2 277.7522} C_DIS
LIN {X -88.7472,Y 14.2559,Z 91,A 165.3259,B 24.9183,C -2.0873,E1 24.8421,E2 279.7688} C_DIS
LIN {X -87.808,Y 19.2035,Z 91,A 162.0687,B 24.9176,C -2.0962,E1 24.8439,E2 283.024} C_DIS
LIN {X -87.1434,Y 22.0263,Z 91,A 160.3135,B 24.9169,C -2.1047,E1 24.845,E2 284.7691} C_DIS
LIN {X -86.246,Y 25.3121,Z 91,A 157.5632,B 24.9177,C -2.0948,E1 24.8472,E2 287.5589} C_DIS
LIN {X -85.1961,Y 28.6469,Z 91,A 155.4346,B 24.9169,C -2.1046,E1 24.8491,E2 289.6764} C_DIS
LIN {X -83.5252,Y 33.2047,Z 91,A 152.6853,B 24.9154,C -2.1241,E1 24.8518,E2 292.3947} C_DIS
LIN {X -81.0296,Y 38.9002,Z 91,A 149.0107,B 24.9138,C -2.1444,E1 24.856,E2 296.041} C_DIS
LIN {X -79.9559,Y 41.0623,Z 91,A 146.6922,B 24.9152,C -2.1262,E1 24.859,E2 298.4152} C_DIS
LIN {X -78.3418,Y 44.0634,Z 91,A 145.119,B 24.9133,C -2.1499,E1 24.861,E2 299.9401} C_DIS
LIN {X -75.7005,Y 48.4609,Z 91,A 141.7466,B 24.9128,C -2.1562,E1 24.8659,E2 303.3149} C_DIS
LIN {X -74.4672,Y 50.3354,Z 91,A 139.9751,B 24.9133,C -2.1502,E1 24.8687,E2 305.1096} C_DIS
LIN {X -71.7892,Y 54.0865,Z 91,A 137.32,B 24.912,C -2.1664,E1 24.8731,E2 307.7389} C_DIS
LIN {X -68.2729,Y 58.4626,Z 91,A 134.1095,B 24.9103,C -2.1865,E1 24.8787,E2 310.9162} C_DIS
LIN {X -64.8285,Y 62.2601,Z 91,A 130.6826,B 24.91,C -2.1899,E1 24.8852,E2 314.3501} C_DIS
LIN {X -60.8002,Y 66.1994,Z 91,A 127.3154,B 24.9088,C -2.2051,E1 24.8919,E2 317.6952} C_DIS
LIN {X -57.3381,Y 69.2198,Z 91,A 124.0514,B 24.9091,C -2.2016,E1 24.8988,E2 320.9803} C_DIS
LIN {X -55.4437,Y 70.7462,Z 91,A 121.6038,B 24.911,C -2.1782,E1 24.9043,E2 323.4927} C_DIS
LIN {X -52.1197,Y 73.2296,Z 91,A 120.1414,B 24.9076,C -2.219,E1 24.9074,E2 324.8631} C_DIS
LIN {X -49.9221,Y 74.7461,Z 91,A 118.0005,B 24.9085,C -2.209,E1 24.9124,E2 327.035} C_DIS
LIN {X -47.5789,Y 76.2579,Z 91,A 115.9647,B 24.9088,C -2.2046,E1 24.9172,E2 329.0878} C_DIS
LIN {X -42.928,Y 78.9697,Z 91,A 111.7185,B 24.9104,C -2.1862,E1 24.9277,E2 333.3901} C_DIS
LIN {X -38.3611,Y 81.2863,Z 91,A 109.2882,B 24.9079,C -2.2164,E1 24.9337,E2 335.7548} C_DIS
LIN {X -35.7677,Y 82.4604,Z 91,A 107.68,B 24.9071,C -2.2253,E1 24.9377,E2 337.3455} C_DIS
LIN {X -31.2255,Y 84.2849,Z 91,A 104.6053,B 24.9066,C -2.2309,E1 24.9457,E2 340.4135} C_DIS
LIN {X -27.0955,Y 85.7025,Z 91,A 101.739,B 24.9066,C -2.2317,E1 24.9533,E2 343.2833} C_DIS
LIN {X -24.2299,Y 86.5564,Z 91,A 99.1022,B 24.9083,C -2.2112,E1 24.9606,E2 345.973} C_DIS
LIN {X -20.3362,Y 87.5518,Z 91,A 97.0106,B 24.9069,C -2.2281,E1 24.9661,E2 348.0273} C_DIS
LIN {X -16.2325,Y 88.4061,Z 91,A 94.5179,B 24.9062,C -2.2358,E1 24.9729,E2 350.5044} C_DIS
LIN {X -12.0413,Y 89.0736,Z 91,A 92.0011,B 24.9056,C -2.2436,E1 24.9798,E2 353.005} C_DIS
LIN {X -9.0122,Y 89.4307,Z 91,A 89.9513,B 24.9058,C -2.2413,E1 24.9855,E2 355.0614} C_DIS
LIN {X -5.6074,Y 89.709,Z 91,A 87.1624,B 24.9073,C -2.2229,E1 24.9934,E2 357.895} C_DIS
LIN {X -2.0171,Y 89.8613,Z 91,A 85.0721,B 24.9067,C -2.2299,E1 24.9992,E2 359.9691} C_DIS
LIN {X 2.7064,Y 89.8426,Z 91,A 82.4172,B 24.9057,C -2.2416,E1 25.0065,E2 362.5956} C_DIS
LIN {X 6.2642,Y 89.665,Z 91,A 79.3443,B 24.9079,C -2.216,E1 25.0153,E2 365.728} C_DIS
LIN {X 10.6688,Y 89.2482,Z 91,A 77.2614,B 24.9059,C -2.2392,E1 25.0209,E2 367.7545} C_DIS
LIN {X 14.3254,Y 88.7358,Z 91,A 74.9199,B 24.9059,C -2.2389,E1 25.0274,E2 370.0945} C_DIS
LIN {X 17.6717,Y 88.1293,Z 91,A 72.8059,B 24.9059,C -2.2397,E1 25.0331,E2 372.204} C_DIS
LIN {X 20.4351,Y 87.5298,Z 91,A 70.9864,B 24.906,C -2.2383,E1 25.0381,E2 374.0245} C_DIS
LIN {X 24.211,Y 86.5618,Z 91,A 67.7295,B 24.9083,C -2.2115,E1 25.047,E2 377.3397} C_DIS
LIN {X 28.4159,Y 85.2736,Z 91,A 65.8458,B 24.9059,C -2.2394,E1 25.0519,E2 379.1538} C_DIS
LIN {X 33.3011,Y 83.4866,Z 91,A 62.3569,B 24.9067,C -2.2305,E1 25.061,E2 382.6562} C_DIS
LIN {X 35.6774,Y 82.4998,Z 91,A 60.7896,B 24.9067,C -2.2311,E1 25.065,E2 384.2182} C_DIS
LIN {X 38.8286,Y 81.064,Z 91,A 57.4158,B 24.91,C -2.1899,E1 25.0738,E2 387.6809} C_DIS
LIN {X 43.8482,Y 78.4624,Z 91,A 55.5096,B 24.9057,C -2.2417,E1 25.0781,E2 389.4589} C_DIS
LIN {X 46.3999,Y 76.9817,Z 91,A 52.6632,B 24.9087,C -2.2063,E1 25.0851,E2 392.3803} C_DIS
LIN {X 49.1441,Y 75.2595,Z 91,A 51.342,B 24.9069,C -2.2282,E1 25.0881,E2 393.6454} C_DIS
LIN {X 53.1245,Y 72.5037,Z 91,A 47.3978,B 24.9097,C -2.194,E1 25.0972,E2 397.657} C_DIS
LIN {X 56.0871,Y 70.2382,Z 91,A 45.9388,B 24.9075,C -2.2209,E1 25.1003,E2 399.0469} C_DIS
LIN {X 61.7633,Y 65.3022,Z 91,A 40.776,B 24.9093,C -2.1988,E1 25.1112,E2 404.2414} C_DIS
LIN {X 64.1954,Y 62.9132,Z 91,A 37.6508,B 24.9124,C -2.1616,E1 25.1174,E2 407.4412} C_DIS
LIN {X 67.6991,Y 59.1258,Z 91,A 35.6708,B 24.9093,C -2.1992,E1 25.1209,E2 409.3236} C_DIS
LIN {X 69.0416,Y 57.5525,Z 91,A 33.8811,B 24.9109,C -2.1798,E1 25.1242,E2 411.151} C_DIS
LIN {X 71.2903,Y 54.7424,Z 91,A 31.9333,B 24.9103,C -2.1863,E1 25.1275,E2 413.0742} C_DIS
LIN {X 73.1814,Y 52.1872,Z 91,A 29.1691,B 24.9128,C -2.1556,E1 25.1321,E2 415.8974} C_DIS
LIN {X 75.3468,Y 49.01,Z 91,A 26.9266,B 24.9128,C -2.1566,E1 25.1355,E2 418.1266} C_DIS
LIN {X 77.6125,Y 45.338,Z 91,A 24.1789,B 24.9134,C -2.1493,E1 25.1395,E2 420.8772} C_DIS
LIN {X 79.5834,Y 41.7794,Z 91,A 22.0882,B 24.9125,C -2.1599,E1 25.1422,E2 422.9319} C_DIS
LIN {X 81.156,Y 38.6353,Z 91,A 19.53,B 24.9139,C -2.1425,E1 25.1453,E2 425.5175} C_DIS
LIN {X 83.2089,Y 33.9891,Z 91,A 16.3017,B 24.9146,C -2.1336,E1 25.1488,E2 428.7493} C_DIS
LIN {X 84.4976,Y 30.6465,Z 91,A 13.3141,B 24.9171,C -2.1021,E1 25.1518,E2 431.7943} C_DIS
LIN {X 86.1151,Y 25.7535,Z 91,A 11.2036,B 24.9146,C -2.1337,E1 25.1534,E2 433.8184} C_DIS
LIN {X 86.8423,Y 23.1841,Z 91,A 9.4347,B 24.9152,C -2.1261,E1 25.1547,E2 435.595} C_DIS
LIN {X 87.661,Y 19.8652,Z 91,A 7.1514,B 24.9161,C -2.1157,E1 25.1562,E2 437.8896} C_DIS
LIN {X 88.2759,Y 16.923,Z 91,A 5.288,B 24.9164,C -2.1116,E1 25.1572,E2 439.7516} C_DIS
LIN {X 88.8394,Y 13.6597,Z 91,A 2.9957,B 24.9174,C -2.0986,E1 25.1582,E2 442.0613} C_DIS
LIN {X 89.4529,Y 8.7911,Z 91,A 0.1043,B 24.9175,C -2.0971,E1 25.1592,E2 444.9391} C_DIS
LIN {X 89.7171,Y 5.4867,Z 91,A -2.0288,B 24.9181,C -2.0897,E1 25.1596,E2 447.0771} C_DIS
LIN {X 89.8801,Y 0.8,Z 91,A -4.6659,B 24.9179,C -2.0928,E1 25.1598,E2 449.6912} C_DIS
LIN {X 89.8083,Y -3.6768,Z 91,A -7.4445,B 24.9184,C -2.0863,E1 25.1597,E2 452.4686} C_DIS
LIN {X 89.5859,Y -7.3075,Z 91,A -10.542,B 24.9211,C -2.051,E1 25.159,E2 455.631} C_DIS
LIN {X 88.9847,Y -12.6787,Z 91,A -13.5112,B 24.9207,C -2.0569,E1 25.158,E2 458.5687} C_DIS
LIN {X 88.0369,Y -18.1252,Z 91,A -16.7824,B 24.9208,C -2.0547,E1 25.1564,E2 461.8259} C_DIS
LIN {X 87.6037,Y -20.1149,Z 91,A -18.8458,B 24.9232,C -2.0233,E1 25.155,E2 463.9515} C_DIS
LIN {X 86.7476,Y -23.5349,Z 91,A -20.5527,B 24.9223,C -2.0354,E1 25.1538,E2 465.6199} C_DIS
LIN {X 85.4218,Y -27.9668,Z 91,A -23.4104,B 24.9228,C -2.0295,E1 25.1515,E2 468.4754} C_DIS
LIN {X 84.374,Y -30.9853,Z 91,A -25.4852,B 24.9234,C -2.0218,E1 25.1495,E2 470.5567} C_DIS
LIN {X 82.2506,Y -36.2477,Z 91,A -28.7569,B 24.9233,C -2.0231,E1 25.1461,E2 473.8072} C_DIS
LIN {X 80.5698,Y -39.8431,Z 91,A -31.5884,B 24.9246,C -2.0048,E1 25.1427,E2 476.6668} C_DIS
LIN {X 79.4846,Y -41.967,Z 91,A -33.9104,B 24.9271,C -1.9719,E1 25.1396,E2 479.0541} C_DIS
LIN {X 77.329,Y -45.8176,Z 91,A -35.6494,B 24.9249,C -2.0018,E1 25.1372,E2 480.7136} C_DIS
LIN {X 74.5753,Y -50.1758,Z 91,A -38.9386,B 24.9256,C -1.9924,E1 25.1323,E2 484.0085} C_DIS
LIN {X 71.9976,Y -53.809,Z 91,A -42.0897,B 24.927,C -1.9736,E1 25.1271,E2 487.1887} C_DIS
LIN {X 68.9103,Y -57.7095,Z 91,A -44.9551,B 24.9268,C -1.976,E1 25.1221,E2 490.0351} C_DIS
LIN {X 67.3973,Y -59.4713,Z 91,A -46.8233,B 24.9281,C -1.9585,E1 25.1186,E2 491.9362} C_DIS
LIN {X 63.4769,Y -63.6387,Z 91,A -50.772,B 24.9295,C -1.939,E1 25.1109,E2 495.9139} C_DIS
LIN {X 60.997,Y -66.0186,Z 91,A -52.4449,B 24.9286,C -1.952,E1 25.1075,E2 497.5495} C_DIS
LIN {X 57.6803,Y -68.9348,Z 91,A -55.6084,B 24.9299,C -1.9335,E1 25.1007,E2 500.7443} C_DIS
LIN {X 53.5081,Y -72.2223,Z 91,A -58.6929,B 24.9297,C -1.9367,E1 25.0939,E2 503.8099} C_DIS
LIN {X 50.5602,Y -74.3151,Z 91,A -61.8629,B 24.9322,C -1.9023,E1 25.0865,E2 507.0504} C_DIS
LIN {X 46.3486,Y -77.0128,Z 91,A -63.6899,B 24.9292,C -1.9432,E1 25.0824,E2 508.7751} C_DIS
LIN {X 41.4235,Y -79.7696,Z 91,A -67.3764,B 24.9299,C -1.9337,E1 25.0734,E2 512.4732} C_DIS
LIN {X 39.3225,Y -80.8257,Z 91,A -69.617,B 24.9319,C -1.9059,E1 25.0676,E2 514.7736} C_DIS
LIN {X 36.3549,Y -82.2029,Z 91,A -71.1124,B 24.9307,C -1.9228,E1 25.0639,E2 516.2252} C_DIS
LIN {X 34.2127,Y -83.1175,Z 91,A -72.5249,B 24.9307,C -1.9231,E1 25.0603,E2 517.6337} C_DIS
LIN {X 31.5425,Y -84.1673,Z 91,A -74.9541,B 24.9323,C -1.9003,E1 25.0538,E2 520.1118} C_DIS
LIN {X 26.851,Y -85.7791,Z 91,A -78.3681,B 24.9332,C -1.888,E1 25.0447,E2 523.5484} C_DIS
LIN {X 22.9839,Y -86.8955,Z 91,A -79.9947,B 24.9311,C -1.9168,E1 25.0405,E2 525.1041} C_DIS
LIN {X 20.4235,Y -87.5325,Z 91,A -81.9433,B 24.9319,C -1.9062,E1 25.0351,E2 527.0751} C_DIS
LIN {X 16.9561,Y -88.2695,Z 91,A -84.1405,B 24.9319,C -1.9063,E1 25.0291,E2 529.2693} C_DIS
LIN {X 13.6991,Y -88.8333,Z 91,A -86.59,B 24.9328,C -1.8934,E1 25.0223,E2 531.7471} C_DIS
LIN {X 8.854,Y -89.4466,Z 91,A -89.4866,B 24.9324,C -1.8987,E1 25.0143,E2 534.629} C_DIS
LIN {X 5.1119,Y -89.738,Z 91,A -91.7696,B 24.9322,C -1.9012,E1 25.0079,E2 536.9049} C_DIS
LIN {X 0.5864,Y -89.8639,Z 91,A -93.6839,B 24.93,C -1.9329,E1 25.0029,E2 538.7437} C_DIS
Enddeposition()
LIN {X 0.5864,Y -89.8639,Z 91,A -93.6839,B 24.93,C -1.9329,E1 25.0029,E2 538.7437} C_DIS
Startdeposition()
$VEL.CP = VEL_PRINT
LIN {X 2.7236,Y -88.8737,Z 91,A -92.3357,B 24.9288,C -1.9487,E1 25.0067,E2 537.3582} C_DIS
LIN {X 6.1696,Y -88.7013,Z 91,A -90.0815,B 24.9287,C -1.9507,E1 25.013,E2 535.1002} C_DIS
LIN {X 8.9527,Y -88.4639,Z 91,A -88.0026,B 24.9279,C -1.961,E1 25.0188,E2 532.9982} C_DIS
LIN {X 13.4627,Y -87.8905,Z 91,A -85.4795,B 24.9288,C -1.9493,E1 25.0257,E2 530.505} C_DIS
LIN {X 16.2695,Y -87.4151,Z 91,A -83.4225,B 24.9281,C -1.9583,E1 25.0314,E2 528.4291} C_DIS
LIN {X 19.4934,Y -86.7526,Z 91,A -81.3635,B 24.9281,C -1.9581,E1 25.037,E2 526.3731} C_DIS
LIN {X 22.7296,Y -85.9616,Z 91,A -78.6812,B 24.9266,C -1.9786,E1 25.0444,E2 523.6464} C_DIS
LIN {X 26.2736,Y -84.945,Z 91,A -76.9342,B 24.928,C -1.9598,E1 25.0489,E2 521.9471} C_DIS
LIN {X 31.1303,Y -83.2878,Z 91,A -73.5639,B 24.9275,C -1.9662,E1 25.0578,E2 518.5684} C_DIS
LIN {X 34.4407,Y -81.9744,Z 91,A -71.4882,B 24.9278,C -1.9619,E1 25.0632,E2 516.5076} C_DIS
LIN {X 37.0712,Y -80.8186,Z 91,A -69.1676,B 24.9264,C -1.9809,E1 25.0692,E2 514.1478} C_DIS
LIN {X 40.7505,Y -79.0282,Z 91,A -66.4164,B 24.9258,C -1.9893,E1 25.076,E2 511.3843} C_DIS
LIN {X 46.5494,Y -75.758,Z 91,A -62.8445,B 24.9271,C -1.972,E1 25.0846,E2 507.8642} C_DIS
LIN {X 49.8156,Y -73.6503,Z 91,A -60.1846,B 24.9263,C -1.9823,E1 25.0908,E2 505.1888} C_DIS
LIN {X 52.1186,Y -72.0399,Z 91,A -58.174,B 24.9255,C -1.9929,E1 25.0954,E2 503.1599} C_DIS
LIN {X 54.6372,Y -70.1495,Z 91,A -56.2767,B 24.9255,C -1.9926,E1 25.0996,E2 501.2703} C_DIS
LIN {X 58.8135,Y -66.6867,Z 91,A -52.7738,B 24.9249,C -2.0007,E1 25.1071,E2 497.7618} C_DIS
LIN {X 61.2697,Y -64.4368,Z 91,A -50.5316,B 24.9243,C -2.0091,E1 25.1117,E2 495.5089} C_DIS
LIN {X 64.2224,Y -61.4937,Z 91,A -47.4627,B 24.9228,C -2.0294,E1 25.1177,E2 492.4054} C_DIS
LIN {X 66.5618,Y -58.9547,Z 91,A -45.7828,B 24.9238,C -2.0156,E1 25.1208,E2 490.7655} C_DIS
LIN {X 69.2113,Y -55.8194,Z 91,A -43.2763,B 24.9237,C -2.0176,E1 25.1252,E2 488.2659} C_DIS
LIN {X 70.5769,Y -54.0824,Z 91,A -40.8602,B 24.9207,C -2.0569,E1 25.1295,E2 485.7682} C_DIS
LIN {X 73.2921,Y -50.3435,Z 91,A -38.85,B 24.9227,C -2.0304,E1 25.1326,E2 483.8306} C_DIS
LIN {X 75.5064,Y -46.955,Z 91,A -36.1643,B 24.9219,C -2.0405,E1 25.1366,E2 481.1345} C_DIS
LIN {X 77.7081,Y -43.2135,Z 91,A -33.1124,B 24.9206,C -2.0577,E1 25.1409,E2 478.0578} C_DIS
LIN {X 79.373,Y -40.0734,Z 91,A -30.9715,B 24.9205,C -2.0591,E1 25.1436,E2 475.925} C_DIS
LIN {X 81.6067,Y -35.3039,Z 91,A -27.3267,B 24.919,C -2.0784,E1 25.1478,E2 472.2545} C_DIS
LIN {X 83.4512,Y -30.6903,Z 91,A -24.6626,B 24.9197,C -2.0688,E1 25.1504,E2 469.6277} C_DIS
LIN {X 84.479,Y -27.7351,Z 91,A -22.5475,B 24.919,C -2.0786,E1 25.1523,E2 467.5014} C_DIS
LIN {X 85.6607,Y -23.8394,Z 91,A -20.2111,B 24.9191,C -2.0765,E1 25.1542,E2 465.1833} C_DIS
LIN {X 86.3021,Y -21.399,Z 91,A -18.0402,B 24.9172,C -2.1013,E1 25.1557,E2 462.9664} C_DIS
LIN {X 87.3292,Y -16.7199,Z 91,A -15.033,B 24.9166,C -2.1083,E1 25.1574,E2 459.9604} C_DIS
LIN {X 88.0951,Y -12.0581,Z 91,A -12.2629,B 24.9166,C -2.1081,E1 25.1585,E2 457.207} C_DIS
LIN {X 88.5221,Y -8.357,Z 91,A -9.8627,B 24.916,C -2.1158,E1 25.1592,E2 454.8028} C_DIS
LIN {X 88.7882,Y -4.7589,Z 91,A -7.6858,B 24.9159,C -2.1179,E1 25.1596,E2 452.6338} C_DIS
LIN {X 88.8721,Y -2.7771,Z 91,A -5.9834,B 24.9143,C -2.1373,E1 25.1598,E2 450.8958} C_DIS
LIN {X 88.9119,Y 0.8483,Z 91,A -3.8434,B 24.9143,C -2.1377,E1 25.1598,E2 448.7676} C_DIS
LIN {X 88.8099,Y 4.3356,Z 91,A -1.7809,B 24.9143,C -2.1382,E1 25.1595,E2 446.7162} C_DIS
LIN {X 88.6173,Y 7.2778,Z 91,A 0.0765,B 24.9139,C -2.1427,E1 25.1591,E2 444.8592} C_DIS
LIN {X 88.4144,Y 9.4278,Z 91,A 1.4991,B 24.9134,C -2.1482,E1 25.1587,E2 443.4319} C_DIS
LIN {X 87.9869,Y 12.8188,Z 91,A 3.5522,B 24.9134,C -2.1498,E1 25.158,E2 441.3873} C_DIS
LIN {X 87.5656,Y 15.436,Z 91,A 5.3842,B 24.9125,C -2.1596,E1 25.1571,E2 439.5429} C_DIS
LIN {X 86.9967,Y 18.3735,Z 91,A 7.3681,B 24.9119,C -2.1675,E1 25.156,E2 437.5518} C_DIS
LIN {X 86.1792,Y 21.89,Z 91,A 9.6564,B 24.9114,C -2.1733,E1 25.1545,E2 435.2631} C_DIS
LIN {X 85.1899,Y 25.4692,Z 91,A 12.441,B 24.9097,C -2.1946,E1 25.1523,E2 432.4442} C_DIS
LIN {X 83.5431,Y 30.4387,Z 91,A 15.3496,B 24.9102,C -2.1879,E1 25.1497,E2 429.5677} C_DIS
LIN {X 82.5819,Y 32.9568,Z 91,A 17.6458,B 24.9081,C -2.2129,E1 25.1472,E2 427.2251} C_DIS
LIN {X 81.2152,Y 36.1942,Z 91,A 19.4031,B 24.9091,C -2.2013,E1 25.1453,E2 425.505} C_DIS
LIN {X 79.8449,Y 39.1244,Z 91,A 21.3578,B 24.9091,C -2.2025,E1 25.1429,E2 423.5579} C_DIS
LIN {X 78.4008,Y 41.9454,Z 91,A 23.343,B 24.9087,C -2.2061,E1 25.1404,E2 421.5748} C_DIS
LIN {X 76.7677,Y 44.8651,Z 91,A 25.6414,B 24.9078,C -2.2169,E1 25.1372,E2 419.2627} C_DIS
LIN {X 74.2212,Y 48.961,Z 91,A 29.1263,B 24.906,C -2.2382,E1 25.1319,E2 415.7448} C_DIS
LIN {X 71.3728,Y 53.0288,Z 91,A 31.9142,B 24.9066,C -2.2316,E1 25.1274,E2 412.9861} C_DIS
LIN {X 67.5592,Y 57.8079,Z 91,A 36.242,B 24.9047,C -2.2545,E1 25.1196,E2 408.6243} C_DIS
LIN {X 62.894,Y 62.8536,Z 91,A 40.3056,B 24.9049,C -2.2513,E1 25.1119,E2 404.5857} C_DIS
LIN {X 59.2331,Y 66.313,Z 91,A 43.9808,B 24.9031,C -2.2728,E1 25.1042,E2 400.8746} C_DIS
LIN {X 56.5216,Y 68.6399,Z 91,A 46.2877,B 24.9027,C -2.2773,E1 25.0992,E2 398.566} C_DIS
LIN {X 53.7253,Y 70.8496,Z 91,A 48.7272,B 24.9019,C -2.2863,E1 25.0938,E2 396.1139} C_DIS
LIN {X 50.3999,Y 73.253,Z 91,A 50.6693,B 24.9036,C -2.2665,E1 25.0895,E2 394.2252} C_DIS
LIN {X 47.9616,Y 74.8709,Z 91,A 53.2679,B 24.9013,C -2.2939,E1 25.0832,E2 391.5703} C_DIS
LIN {X 44.392,Y 77.041,Z 91,A 55.1655,B 24.9033,C -2.2707,E1 25.0788,E2 389.7334} C_DIS
LIN {X 42.5442,Y 78.0767,Z 91,A 57.3974,B 24.9006,C -2.302,E1 25.0731,E2 387.4338} C_DIS
LIN {X 38.5801,Y 80.1096,Z 91,A 59.3845,B 24.9029,C -2.2755,E1 25.0683,E2 385.5145} C_DIS
LIN {X 35.9149,Y 81.3393,Z 91,A 61.258,B 24.9027,C -2.2771,E1 25.0635,E2 383.6421} C_DIS
LIN {X 33.8443,Y 82.2225,Z 91,A 62.6594,B 24.9027,C -2.277,E1 25.0599,E2 382.2443} C_DIS
LIN {X 29.9993,Y 83.7024,Z 91,A 65.4353,B 24.9022,C -2.2835,E1 25.0527,E2 379.4588} C_DIS
LIN {X 26.9247,Y 84.7416,Z 91,A 67.3062,B 24.9027,C -2.2779,E1 25.0477,E2 377.6048} C_DIS
LIN {X 23.6297,Y 85.7184,Z 91,A 69.4576,B 24.9027,C -2.2773,E1 25.042,E2 375.4584} C_DIS
LIN {X 20.4802,Y 86.5247,Z 91,A 71.788,B 24.9019,C -2.2863,E1 25.0356,E2 373.1101} C_DIS
LIN {X 17.1436,Y 87.2478,Z 91,A 74.059,B 24.9016,C -2.2896,E1 25.0294,E2 370.8341} C_DIS
LIN {X 13.8747,Y 87.8268,Z 91,A 76.1078,B 24.9018,C -2.2874,E1 25.0238,E2 368.7927} C_DIS
LIN {X 10.4859,Y 88.2951,Z 91,A 78.0968,B 24.9024,C -2.2809,E1 25.0183,E2 366.8208} C_DIS
LIN {X 6.6366,Y 88.6685,Z 91,A 80.7936,B 24.9018,C -2.2877,E1 25.0108,E2 364.1093} C_DIS
LIN {X 3.6701,Y 88.8398,Z 91,A 82.7016,B 24.9018,C -2.2874,E1 25.0055,E2 362.2026} C_DIS
LIN {X 0.6744,Y 88.913,Z 91,A 84.3491,B 24.9026,C -2.2781,E1 25.0009,E2 360.5775} C_DIS
LIN {X -2.241,Y 88.8872,Z 91,A 86.8728,B 24.9009,C -2.2983,E1 24.9937,E2 358.0057} C_DIS
LIN {X -6.7577,Y 88.6589,Z 91,A 89.4684,B 24.9019,C -2.2869,E1 24.9866,E2 355.4362} C_DIS
LIN {X -10.2099,Y 88.3274,Z 91,A 91.7219,B 24.9019,C -2.2863,E1 24.9803,E2 353.1828} C_DIS
LIN {X -14.7578,Y 87.6822,Z 91,A 94.6623,B 24.9022,C -2.2837,E1 24.9722,E2 350.246} C_DIS
LIN {X -17.9288,Y 87.0892,Z 91,A 97.2916,B 24.9008,C -2.2994,E1 24.9649,E2 347.5764} C_DIS
LIN {X -21.2912,Y 86.329,Z 91,A 99.5648,B 24.9008,C -2.2989,E1 24.9587,E2 345.3012} C_DIS
LIN {X -24.7368,Y 85.405,Z 91,A 101.214,B 24.9028,C -2.2761,E1 24.9544,E2 343.7036} C_DIS
LIN {X -29.6164,Y 83.8383,Z 91,A 104.8448,B 24.9023,C -2.2823,E1 24.9448,E2 340.0513} C_DIS
LIN {X -34.1438,Y 82.0983,Z 91,A 107.5604,B 24.9037,C -2.2654,E1 24.9378,E2 337.37} C_DIS
LIN {X -36.5895,Y 81.0381,Z 91,A 109.4174,B 24.9036,C -2.2671,E1 24.933,E2 335.5044} C_DIS
LIN {X -41.1208,Y 78.8357,Z 91,A 112.7293,B 24.9038,C -2.2639,E1 24.9248,E2 332.1914} C_DIS
LIN {X -44.0907,Y 77.2142,Z 91,A 114.6124,B 24.9049,C -2.2511,E1 24.9202,E2 330.3334} C_DIS
LIN {X -45.6798,Y 76.2856,Z 91,A 116.0615,B 24.9044,C -2.2569,E1 24.9167,E2 328.866} C_DIS
LIN {X -50.1696,Y 73.4101,Z 91,A 119.5234,B 24.9049,C -2.2512,E1 24.9086,E2 325.4066} C_DIS
LIN {X -53.4527,Y 71.0547,Z 91,A 122.4909,B 24.9045,C -2.2568,E1 24.9019,E2 322.4151} C_DIS
LIN {X -57.6949,Y 67.6555,Z 91,A 126.0613,B 24.9049,C -2.2512,E1 24.8942,E2 318.8445} C_DIS
LIN {X -60.1447,Y 65.4873,Z 91,A 128.2813,B 24.9051,C -2.2497,E1 24.8896,E2 316.6192} C_DIS
LIN {X -62.4944,Y 63.2488,Z 91,A 129.8875,B 24.9067,C -2.2301,E1 24.8865,E2 315.0528} C_DIS
LIN {X -65.1599,Y 60.5002,Z 91,A 132.8678,B 24.9059,C -2.2394,E1 24.8807,E2 312.0375} C_DIS
LIN {X -67.3566,Y 58.0457,Z 91,A 134.9663,B 24.9064,C -2.2332,E1 24.8769,E2 309.944} C_DIS
LIN {X -69.8665,Y 54.997,Z 91,A 137.2725,B 24.9076,C -2.2195,E1 24.8729,E2 307.6599} C_DIS
LIN {X -73.2278,Y 50.4346,Z 91,A 140.6219,B 24.9092,C -2.2006,E1 24.8675,E2 304.3391} C_DIS
LIN {X -74.3958,Y 48.6961,Z 91,A 142.3255,B 24.9086,C -2.2073,E1 24.8649,E2 302.6111} C_DIS
LIN {X -77.1691,Y 44.1691,Z 91,A 146.0935,B 24.9086,C -2.2078,E1 24.8595,E2 298.8224} C_DIS
LIN {X -78.8212,Y 41.1485,Z 91,A 147.8045,B 24.9103,C -2.1863,E1 24.8573,E2 297.1536} C_DIS
LIN {X -80.3121,Y 38.1561,Z 91,A 149.882,B 24.911,C -2.1777,E1 24.8548,E2 295.0854} C_DIS
LIN {X -82.5094,Y 33.138,Z 91,A 153.5053,B 24.9117,C -2.1697,E1 24.8508,E2 291.461} C_DIS
LIN {X -84.7537,Y 26.8861,Z 91,A 157.8933,B 24.9125,C -2.1596,E1 24.8468,E2 287.0723} C_DIS
LIN {X -85.7335,Y 23.5746,Z 91,A 160.0551,B 24.9132,C -2.1508,E1 24.8451,E2 284.919} C_DIS
LIN {X -86.514,Y 20.525,Z 91,A 162.1851,B 24.9135,C -2.1474,E1 24.8437,E2 282.7847} C_DIS
LIN {X -87.0512,Y 18.1138,Z 91,A 164.1512,B 24.913,C -2.1533,E1 24.8426,E2 280.793} C_DIS
LIN {X -87.9017,Y 13.3899,Z 91,A 166.4817,B 24.9156,C -2.1212,E1 24.8415,E2 278.5253} C_DIS
LIN {X -88.4446,Y 9.1395,Z 91,A 169.5477,B 24.9156,C -2.1212,E1 24.8405,E2 275.441} C_DIS
LIN {X -88.8833,Y 2.3933,Z 91,A 173.8706,B 24.9168,C -2.1061,E1 24.8398,E2 271.1279} C_DIS
LIN {X -88.906,Y -1.309,Z 91,A 176.4827,B 24.9168,C -2.1051,E1 24.8398,E2 268.5026} C_DIS
LIN {X -88.6081,Y -7.3939,Z 91,A -179.621,B 24.9179,C -2.0917,E1 24.8405,E2 264.6147} C_DIS
LIN {X -87.9352,Y -13.1735,Z 91,A -175.7584,B 24.9186,C -2.0832,E1 24.8419,E2 260.7494} C_DIS
LIN {X -87.1269,Y -17.7447,Z 91,A -173.0609,B 24.92,C -2.0653,E1 24.8432,E2 258.0786} C_DIS
LIN {X -86.5313,Y -20.4529,Z 91,A -170.5278,B 24.9187,C -2.0818,E1 24.8449,E2 255.4913} C_DIS
LIN {X -85.6737,Y -23.792,Z 91,A -169.0629,B 24.921,C -2.0527,E1 24.8459,E2 254.0872} C_DIS
LIN {X -84.7337,Y -26.9497,Z 91,A -166.7297,B 24.921,C -2.0525,E1 24.8478,E2 251.741} C_DIS
LIN {X -83.8485,Y -29.5875,Z 91,A -164.8559,B 24.9212,C -2.0497,E1 24.8495,E2 249.8635} C_DIS
LIN {X -82.4234,Y -33.3524,Z 91,A -162.2212,B 24.9217,C -2.0433,E1 24.8522,E2 247.2291} C_DIS
LIN {X -81.1823,Y -36.2682,Z 91,A -160.1366,B 24.9221,C -2.0388,E1 24.8545,E2 245.1439} C_DIS
LIN {X -79.6033,Y -39.6142,Z 91,A -157.335,B 24.9216,C -2.0446,E1 24.858,E2 242.3132} C_DIS
LIN {X -78.096,Y -42.5088,Z 91,A -155.663,B 24.923,C -2.026,E1 24.8602,E2 240.6767} C_DIS
LIN {X -76.2699,Y -45.7063,Z 91,A -153.1213,B 24.9231,C -2.0248,E1 24.8638,E2 238.1249} C_DIS
LIN {X -74.101,Y -49.1432,Z 91,A -150.7976,B 24.9243,C -2.0092,E1 24.8673,E2 235.8265} C_DIS
LIN {X -71.0487,Y -53.4608,Z 91,A -147.215,B 24.9245,C -2.0061,E1 24.8731,E2 232.234} C_DIS
LIN {X -68.8785,Y -56.2301,Z 91,A -144.959,B 24.925,C -2.0004,E1 24.8771,E2 229.9811} C_DIS
LIN {X -65.3601,Y -60.2832,Z 91,A -141.4506,B 24.9254,C -1.9941,E1 24.8836,E2 226.4719} C_DIS
LIN {X -62.8142,Y -62.9306,Z 91,A -138.1059,B 24.9235,C -2.0192,E1 24.8903,E2 223.053} C_DIS
LIN {X -59.1292,Y -66.406,Z 91,A -135.7812,B 24.9262,C -1.9836,E1 24.895,E2 220.8038} C_DIS
LIN {X -56.7808,Y -68.4244,Z 91,A -133.0402,B 24.9248,C -2.003,E1 24.901,E2 218.0062} C_DIS
LIN {X -53.3941,Y -71.0987,Z 91,A -131.0916,B 24.9271,C -1.9722,E1 24.9052,E2 216.1239} C_DIS
LIN {X -51.1121,Y -72.7574,Z 91,A -128.5676,B 24.9257,C -1.9912,E1 24.911,E2 213.546} C_DIS
LIN {X -47.9499,Y -74.8784,Z 91,A -126.7481,B 24.9274,C -1.9675,E1 24.9152,E2 211.777} C_DIS
LIN {X -44.6401,Y -76.8983,Z 91,A -123.6593,B 24.9263,C -1.9825,E1 24.9227,E2 208.6432} C_DIS
LIN {X -41.4905,Y -78.6416,Z 91,A -121.9572,B 24.928,C -1.96,E1 24.9268,E2 206.99} C_DIS
LIN {X -38.6956,Y -80.0541,Z 91,A -119.8492,B 24.928,C -1.9604,E1 24.9321,E2 204.8755} C_DIS
LIN {X -33.2983,Y -82.4452,Z 91,A -116.0215,B 24.9282,C -1.9571,E1 24.9419,E2 201.0466} C_DIS
LIN {X -29.8522,Y -83.7547,Z 91,A -113.9617,B 24.9291,C -1.9449,E1 24.9472,E2 199.0116} C_DIS
LIN {X -26.6795,Y -84.8186,Z 91,A -111.7385,B 24.9291,C -1.9453,E1 24.9531,E2 196.7833} C_DIS
LIN {X -23.4815,Y -85.7591,Z 91,A -109.435,B 24.9288,C -1.9489,E1 24.9594,E2 194.4676} C_DIS
LIN {X -19.308,Y -86.7944,Z 91,A -106.512,B 24.9285,C -1.9524,E1 24.9673,E2 191.5324} C_DIS
LIN {X -15.7541,Y -87.5087,Z 91,A -104.2831,B 24.9289,C -1.948,E1 24.9734,E2 189.3114} C_DIS
LIN {X -12.1353,Y -88.0843,Z 91,A -101.9358,B 24.9289,C -1.947,E1 24.9799,E2 186.9646} C_DIS
LIN {X -8.9245,Y -88.4668,Z 91,A -99.9143,B 24.9291,C -1.9447,E1 24.9855,E2 184.9472} C_DIS
LIN {X -5.4931,Y -88.7466,Z 91,A -97.6335,B 24.9289,C -1.9467,E1 24.9919,E2 182.6608} C_DIS
LIN {X -0.9943,Y -88.911,Z 91,A -94.9415,B 24.9294,C -1.9402,E1 24.9994,E2 179.9837} C_DIS
LIN {X 0.5714,Y -88.9076,Z 91,A -93.7115,B 24.9289,C -1.9479,E1 25.0028,E2 178.7357} C_DIS
Enddeposition()
LIN {X 0.5714,Y -88.9076,Z 91,A -93.7115,B 24.9289,C -1.9479,E1 25.0028,E2 178.7357} C_DIS
Startdeposition()
$VEL.CP = VEL_PRINT
LIN {X -1.1892,Y -87.9399,Z 91,A -95.9672,B 24.9303,C -1.9283,E1 24.9964,E2 181.0377} C_DIS
LIN {X -4.9204,Y -87.8099,Z 91,A -98.315,B 24.9301,C -1.9308,E1 24.9899,E2 183.3802} C_DIS
LIN {X -8.4071,Y -87.5454,Z 91,A -100.6138,B 24.9301,C -1.9303,E1 24.9835,E2 185.6814} C_DIS
LIN {X -11.8442,Y -87.1471,Z 91,A -102.9088,B 24.9302,C -1.9294,E1 24.9771,E2 187.9802} C_DIS
LIN {X -15.3391,Y -86.5996,Z 91,A -105.1909,B 24.9302,C -1.9308,E1 24.9708,E2 190.2611} C_DIS
LIN {X -18.8967,Y -85.8936,Z 91,A -107.2837,B 24.9294,C -1.9402,E1 24.9652,E2 192.3339} C_DIS
LIN {X -21.0931,Y -85.381,Z 91,A -109.0449,B 24.93,C -1.9319,E1 24.9603,E2 194.1174} C_DIS
LIN {X -26.4731,Y -83.8689,Z 91,A -112.6642,B 24.9298,C -1.935,E1 24.9506,E2 197.7351} C_DIS
LIN {X -29.5524,Y -82.834,Z 91,A -114.7046,B 24.9295,C -1.9391,E1 24.9452,E2 199.7697} C_DIS
LIN {X -32.3655,Y -81.7759,Z 91,A -116.7006,B 24.9295,C -1.9398,E1 24.94,E2 201.7684} C_DIS
LIN {X -35.4967,Y -80.4659,Z 91,A -118.9888,B 24.9295,C -1.9398,E1 24.9341,E2 204.062} C_DIS
LIN {X -38.7971,Y -78.9273,Z 91,A -121.3718,B 24.9293,C -1.9422,E1 24.9281,E2 206.4451} C_DIS
LIN {X -41.3299,Y -77.6323,Z 91,A -123.3078,B 24.9293,C -1.9421,E1 24.9233,E2 208.3869} C_DIS
LIN {X -44.7212,Y -75.7284,Z 91,A -125.6596,B 24.9286,C -1.9511,E1 24.9177,E2 210.7241} C_DIS
LIN {X -47.3366,Y -74.1219,Z 91,A -127.6617,B 24.9284,C -1.9541,E1 24.9129,E2 212.7256} C_DIS
LIN {X -50.2358,Y -72.1882,Z 91,A -130.0421,B 24.9284,C -1.9544,E1 24.9074,E2 215.113} C_DIS
LIN {X -52.687,Y -70.4193,Z 91,A -132.1301,B 24.9284,C -1.9543,E1 24.9027,E2 217.2089} C_DIS
LIN {X -55.7275,Y -68.0393,Z 91,A -134.5704,B 24.9279,C -1.9611,E1 24.8974,E2 219.6421} C_DIS
LIN {X -58.4909,Y -65.6784,Z 91,A -136.5645,B 24.9267,C -1.9768,E1 24.8933,E2 221.6066} C_DIS
LIN {X -62.2832,Y -62.0947,Z 91,A -140.3424,B 24.9271,C -1.9725,E1 24.8856,E2 225.4103} C_DIS
LIN {X -64.038,Y -60.2819,Z 91,A -142.2685,B 24.9274,C -1.9678,E1 24.8819,E2 227.356} C_DIS
LIN {X -66.9166,Y -57.0696,Z 91,A -144.7078,B 24.9261,C -1.985,E1 24.8774,E2 229.7653} C_DIS
LIN {X -68.8659,Y -54.702,Z 91,A -146.6605,B 24.9257,C -1.991,E1 24.874,E2 231.7128} C_DIS
LIN {X -70.5367,Y -52.5307,Z 91,A -148.5007,B 24.9255,C -1.9937,E1 24.8709,E2 233.5555} C_DIS
LIN {X -72.5804,Y -49.6689,Z 91,A -150.9071,B 24.9253,C -1.996,E1 24.867,E2 235.968} C_DIS
LIN {X -74.324,Y -47.0202,Z 91,A -152.9167,B 24.9248,C -2.003,E1 24.864,E2 237.9712} C_DIS
LIN {X -75.7894,Y -44.618,Z 91,A -154.7994,B 24.9245,C -2.0064,E1 24.8613,E2 239.8556} C_DIS
LIN {X -77.3887,Y -41.7828,Z 91,A -157.4422,B 24.9252,C -1.9971,E1 24.8577,E2 242.5343} C_DIS
LIN {X -78.8965,Y -38.8599,Z 91,A -159.0029,B 24.9235,C -2.0197,E1 24.8558,E2 244.0496} C_DIS
LIN {X -80.3753,Y -35.7007,Z 91,A -161.3887,B 24.9233,C -2.0228,E1 24.853,E2 246.4409} C_DIS
LIN {X -81.677,Y -32.6129,Z 91,A -163.5789,B 24.9228,C -2.0289,E1 24.8507,E2 248.6287} C_DIS
LIN {X -82.8724,Y -29.4443,Z 91,A -165.8324,B 24.9224,C -2.034,E1 24.8486,E2 250.8829} C_DIS
LIN {X -83.9845,Y -26.1032,Z 91,A -168.1957,B 24.922,C -2.0389,E1 24.8465,E2 253.2481} C_DIS
LIN {X -84.7601,Y -23.4638,Z 91,A -170.9254,B 24.9236,C -2.018,E1 24.8445,E2 256.0436} C_DIS
LIN {X -85.9481,Y -18.6468,Z 91,A -172.9034,B 24.9202,C -2.0632,E1 24.8433,E2 257.9253} C_DIS
LIN {X -86.4264,Y -16.2876,Z 91,A -174.7778,B 24.9205,C -2.0593,E1 24.8423,E2 259.82} C_DIS
LIN {X -86.9738,Y -13.0568,Z 91,A -177.0731,B 24.9203,C -2.0614,E1 24.8413,E2 262.1239} C_DIS
LIN {X -87.5672,Y -8.171,Z 91,A -179.7592,B 24.9184,C -2.0863,E1 24.8405,E2 264.7668} C_DIS
LIN {X -87.7957,Y -5.1665,Z 91,A 177.7847,B 24.919,C -2.0786,E1 24.84,E2 267.256} C_DIS
LIN {X -87.9457,Y 0.5369,Z 91,A 174.135,B 24.9179,C -2.0923,E1 24.8398,E2 270.8949} C_DIS
LIN {X -87.8728,Y 3.6281,Z 91,A 171.2862,B 24.9192,C -2.0755,E1 24.8401,E2 273.801} C_DIS
LIN {X -87.5816,Y 8.0149,Z 91,A 168.7683,B 24.9177,C -2.0943,E1 24.8407,E2 276.2892} C_DIS
LIN {X -87.2319,Y 11.1975,Z 91,A 166.7175,B 24.9171,C -2.1019,E1 24.8415,E2 278.334} C_DIS
LIN {X -86.701,Y 14.7575,Z 91,A 164.5,B 24.9163,C -2.1129,E1 24.8425,E2 280.5384} C_DIS
LIN {X -85.9037,Y 18.8504,Z 91,A 162.0847,B 24.9149,C -2.13,E1 24.8438,E2 282.9272} C_DIS
LIN {X -85.1759,Y 21.9054,Z 91,A 160.023,B 24.9144,C -2.136,E1 24.8452,E2 284.9866} C_DIS
LIN {X -84.338,Y 24.9375,Z 91,A 157.9325,B 24.914,C -2.1413,E1 24.8468,E2 287.0767} C_DIS
LIN {X -83.3996,Y 27.9162,Z 91,A 156.1755,B 24.9129,C -2.1554,E1 24.8483,E2 288.8099} C_DIS
LIN {X -82.3957,Y 30.7523,Z 91,A 153.8607,B 24.9132,C -2.1514,E1 24.8505,E2 291.1474} C_DIS
LIN {X -80.8503,Y 34.6126,Z 91,A 151.2004,B 24.9124,C -2.161,E1 24.8533,E2 293.7996} C_DIS
LIN {X -79.5726,Y 37.4573,Z 91,A 149.1072,B 24.9121,C -2.1654,E1 24.8558,E2 295.8939} C_DIS
LIN {X -77.9927,Y 40.6442,Z 91,A 146.6228,B 24.9119,C -2.1674,E1 24.8589,E2 298.3866} C_DIS
LIN {X -75.6172,Y 44.9093,Z 91,A 143.1108,B 24.9119,C -2.1672,E1 24.8638,E2 301.9174} C_DIS
LIN {X -73.9232,Y 47.6462,Z 91,A 141.4407,B 24.9104,C -2.1852,E1 24.8663,E2 303.5531} C_DIS
LIN {X -72.3879,Y 49.9485,Z 91,A 139.3197,B 24.9108,C -2.1811,E1 24.8697,E2 305.6944} C_DIS
LIN {X -68.7017,Y 54.9092,Z 91,A 135.6137,B 24.9091,C -2.2009,E1 24.8759,E2 309.3707} C_DIS
LIN {X -66.5164,Y 57.5369,Z 91,A 133.2878,B 24.9089,C -2.2038,E1 24.8801,E2 311.7004} C_DIS
LIN {X -64.2485,Y 60.0581,Z 91,A 131.108,B 24.9084,C -2.2102,E1 24.8842,E2 313.8747} C_DIS
LIN {X -61.9005,Y 62.475,Z 91,A 128.9971,B 24.9077,C -2.2179,E1 24.8883,E2 315.9761} C_DIS
LIN {X -59.0744,Y 65.1549,Z 91,A 126.3334,B 24.9075,C -2.2201,E1 24.8938,E2 318.6454} C_DIS
LIN {X -54.9126,Y 68.699,Z 91,A 122.6844,B 24.9071,C -2.2254,E1 24.9016,E2 322.2958} C_DIS
LIN {X -51.3854,Y 71.375,Z 91,A 120.0606,B 24.906,C -2.239,E1 24.9075,E2 324.8965} C_DIS
LIN {X -48.9269,Y 73.0822,Z 91,A 118.0009,B 24.906,C -2.2396,E1 24.9122,E2 326.9618} C_DIS
LIN {X -46.3247,Y 74.759,Z 91,A 116.0701,B 24.9054,C -2.2459,E1 24.9167,E2 328.8837} C_DIS
LIN {X -43.4857,Y 76.4454,Z 91,A 113.8441,B 24.9052,C -2.2475,E1 24.9221,E2 331.1125} C_DIS
LIN {X -40.9415,Y 77.8368,Z 91,A 111.8789,B 24.9052,C -2.2485,E1 24.927,E2 333.081} C_DIS
LIN {X -37.5793,Y 79.5146,Z 91,A 109.4024,B 24.9049,C -2.2515,E1 24.9332,E2 335.5567} C_DIS
LIN {X -34.4088,Y 80.9375,Z 91,A 107.0478,B 24.9049,C -2.2521,E1 24.9392,E2 337.9155} C_DIS
LIN {X -29.2996,Y 82.9237,Z 91,A 103.6367,B 24.904,C -2.2616,E1 24.9481,E2 341.3112} C_DIS
LIN {X -26.3723,Y 83.9006,Z 91,A 101.512,B 24.9041,C -2.2605,E1 24.9537,E2 343.4423} C_DIS
LIN {X -22.9894,Y 84.8897,Z 91,A 99.3052,B 24.9037,C -2.2656,E1 24.9597,E2 345.6404} C_DIS
LIN {X -17.9447,Y 86.0978,Z 91,A 95.8506,B 24.9037,C -2.2664,E1 24.9691,E2 349.0977} C_DIS
LIN {X -14.6456,Y 86.7196,Z 91,A 93.6295,B 24.9036,C -2.267,E1 24.9752,E2 351.3196} C_DIS
LIN {X -11.751,Y 87.1593,Z 91,A 91.7482,B 24.9034,C -2.269,E1 24.9804,E2 353.1975} C_DIS
LIN {X -8.3363,Y 87.552,Z 91,A 89.5062,B 24.9034,C -2.2701,E1 24.9866,E2 355.4383} C_DIS
LIN {X -4.7603,Y 87.8187,Z 91,A 87.1213,B 24.9034,C -2.2696,E1 24.9932,E2 357.8253} C_DIS
LIN {X -1.0226,Y 87.9425,Z 91,A 84.6839,B 24.9034,C -2.2702,E1 25,E2 360.2615} C_DIS
LIN {X 2.5899,Y 87.9095,Z 91,A 82.3674,B 24.9032,C -2.2716,E1 25.0065,E2 362.5741} C_DIS
LIN {X 5.3204,Y 87.7877,Z 91,A 80.5572,B 24.9032,C -2.2707,E1 25.0115,E2 364.3859} C_DIS
LIN {X 8.6117,Y 87.5254,Z 91,A 78.3976,B 24.9033,C -2.2703,E1 25.0175,E2 366.5453} C_DIS
LIN {X 12.1811,Y 87.1001,Z 91,A 76.1032,B 24.9033,C -2.2713,E1 25.0239,E2 368.8355} C_DIS
LIN {X 15.7868,Y 86.5194,Z 91,A 73.6766,B 24.9034,C -2.269,E1 25.0306,E2 371.265} C_DIS
LIN {X 19.2544,Y 85.8143,Z 91,A 71.7243,B 24.9025,C -2.2791,E1 25.0358,E2 373.1907} C_DIS
LIN {X 23.4454,Y 84.7652,Z 91,A 68.5988,B 24.9035,C -2.2674,E1 25.0444,E2 376.3391} C_DIS
LIN {X 26.5046,Y 83.859,Z 91,A 66.5726,B 24.9035,C -2.2676,E1 25.0498,E2 378.3614} C_DIS
LIN {X 29.3715,Y 82.8983,Z 91,A 64.6334,B 24.9035,C -2.2669,E1 25.0549,E2 380.2985} C_DIS
LIN {X 31.9268,Y 81.9482,Z 91,A 62.8149,B 24.9039,C -2.2638,E1 25.0596,E2 382.1204} C_DIS
LIN {X 35.0951,Y 80.6419,Z 91,A 60.5302,B 24.9042,C -2.2597,E1 25.0655,E2 384.4092} C_DIS
LIN {X 38.3983,Y 79.1231,Z 91,A 58.0269,B 24.9048,C -2.2525,E1 25.0718,E2 386.9232} C_DIS
LIN {X 41.5891,Y 77.4935,Z 91,A 55.8189,B 24.9048,C -2.2536,E1 25.0773,E2 389.1225} C_DIS
LIN {X 45.0297,Y 75.546,Z 91,A 53.1873,B 24.9052,C -2.248,E1 25.0837,E2 391.7592} C_DIS
LIN {X 48.3501,Y 73.4646,Z 91,A 50.787,B 24.9052,C -2.2491,E1 25.0893,E2 394.1492} C_DIS
LIN {X 53.2175,Y 70.0207,Z 91,A 46.8295,B 24.9059,C -2.24,E1 25.0983,E2 398.1142} C_DIS
LIN {X 56.07,Y 67.7567,Z 91,A 44.732,B 24.9055,C -2.2448,E1 25.1028,E2 400.1925} C_DIS
LIN {X 58.7821,Y 65.4177,Z 91,A 41.7132,B 24.9078,C -2.2173,E1 25.1092,E2 403.2643} C_DIS
LIN {X 61.2467,Y 63.1166,Z 91,A 40.2213,B 24.9062,C -2.2364,E1 25.1121,E2 404.705} C_DIS
LIN {X 64.3775,Y 59.9205,Z 91,A 37.0887,B 24.9073,C -2.2227,E1 25.1182,E2 407.8564} C_DIS
LIN {X 66.721,Y 57.2993,Z 91,A 34.8684,B 24.9076,C -2.2199,E1 25.1223,E2 410.0734} C_DIS
LIN {X 69.3245,Y 54.1215,Z 91,A 32.2185,B 24.908,C -2.2144,E1 25.1269,E2 412.7239} C_DIS
LIN {X 71.2426,Y 51.5694,Z 91,A 30.3287,B 24.9079,C -2.2158,E1 25.13,E2 414.6013} C_DIS
LIN {X 73.5523,Y 48.2171,Z 91,A 27.4321,B 24.9092,C -2.2007,E1 25.1346,E2 417.5192} C_DIS
LIN {X 75.2396,Y 45.5391,Z 91,A 25.5625,B 24.9091,C -2.202,E1 25.1373,E2 419.3765} C_DIS
LIN {X 76.8411,Y 42.7811,Z 91,A 23.4798,B 24.9095,C -2.1962,E1 25.1402,E2 421.4619} C_DIS
LIN {X 78.3739,Y 39.9036,Z 91,A 21.3153,B 24.9101,C -2.189,E1 25.143,E2 423.632} C_DIS
LIN {X 79.7929,Y 36.9849,Z 91,A 19.3964,B 24.9101,C -2.1898,E1 25.1453,E2 425.5386} C_DIS
LIN {X 80.9026,Y 34.4904,Z 91,A 17.484,B 24.9108,C -2.1801,E1 25.1475,E2 427.4635} C_DIS
LIN {X 82.0006,Y 31.793,Z 91,A 15.3828,B 24.9119,C -2.1676,E1 25.1497,E2 429.5828} C_DIS
LIN {X 82.9479,Y 29.2307,Z 91,A 13.2181,B 24.9134,C -2.149,E1 25.1517,E2 431.779} C_DIS
LIN {X 84.011,Y 26.0177,Z 91,A 11.7271,B 24.9119,C -2.1671,E1 25.1529,E2 433.2188} C_DIS
LIN {X 84.7306,Y 23.5711,Z 91,A 9.8326,B 24.913,C -2.154,E1 25.1544,E2 435.1335} C_DIS
LIN {X 85.6434,Y 20.0007,Z 91,A 7.4834,B 24.9134,C -2.1485,E1 25.156,E2 437.4822} C_DIS
LIN {X 86.3134,Y 16.8772,Z 91,A 5.4229,B 24.9139,C -2.1427,E1 25.1571,E2 439.5442} C_DIS
LIN {X 86.9358,Y 13.3026,Z 91,A 3.0914,B 24.9144,C -2.1365,E1 25.1582,E2 441.8768} C_DIS
LIN {X 87.3766,Y 10.0077,Z 91,A 0.9057,B 24.915,C -2.1289,E1 25.1589,E2 444.0673} C_DIS
LIN {X 87.7122,Y 6.4513,Z 91,A -1.4559,B 24.9157,C -2.1203,E1 25.1595,E2 446.4352} C_DIS
LIN {X 87.9024,Y 2.8211,Z 91,A -3.4749,B 24.9153,C -2.125,E1 25.1597,E2 448.4311} C_DIS
LIN {X 87.9477,Y 0.1283,Z 91,A -5.5561,B 24.9167,C -2.108,E1 25.1597,E2 450.5403} C_DIS
LIN {X 87.872,Y -3.6469,Z 91,A -7.8973,B 24.917,C -2.1042,E1 25.1596,E2 452.8764} C_DIS
LIN {X 87.6617,Y -7.0851,Z 91,A -10.1258,B 24.9175,C -2.0976,E1 25.1591,E2 455.1074} C_DIS
LIN {X 87.3075,Y -10.5934,Z 91,A -12.4135,B 24.918,C -2.0905,E1 25.1584,E2 457.3981} C_DIS
LIN {X 86.8217,Y -14.0348,Z 91,A -14.5868,B 24.9184,C -2.0865,E1 25.1575,E2 459.5682} C_DIS
LIN {X 85.9639,Y -18.5739,Z 91,A -17.7401,B 24.9195,C -2.0718,E1 25.1558,E2 462.7376} C_DIS
LIN {X 84.8676,Y -23.0712,Z 91,A -20.2761,B 24.9189,C -2.0791,E1 25.1541,E2 465.2417} C_DIS
LIN {X 84.1637,Y -25.521,Z 91,A -22.1988,B 24.9201,C -2.0647,E1 25.1526,E2 467.1876} C_DIS
Enddeposition()
END
